  MoveL 5226 to (-61.59, 2.74, -134.54) mm, rotated rx -172.19 ry 6.28 rz 7.52 deg; joints [-5.137, -27.027, 87, 93.373, 104.768, 50.925, -36.259]
  MoveL 5227 to (-61.07, 2.44, -134.84) mm, rotated rx -172.19 ry 6.28 rz 7.52 deg; joints [-5.158, -27.049, 87.032, 93.353, 104.779, 50.915, -36.259]
  MoveL 5228 to (-60.98, 2.39, -135) mm, rotated rx -172.19 ry 6.28 rz 7.52 deg; joints [-5.162, -27.056, 87.036, 93.35, 104.781, 50.918, -36.259]
  MoveL 5229 to (-61.28, 2.57, -135.03) mm, rotated rx -172.19 ry 6.28 rz 7.52 deg; joints [-5.153, -27.051, 87.016, 93.362, 104.775, 50.934, -36.259]
  MoveL 5230 to (-61.68, 2.81, -135.05) mm, rotated rx -172.19 ry 6.28 rz 7.52 deg; joints [-5.14, -27.044, 86.989, 93.378, 104.768, 50.954, -36.259]
  MoveL 5231 to (-62.08, 3.07, -135.08) mm, rotated rx -172.19 ry 6.28 rz 7.52 deg; joints [-5.127, -27.036, 86.96, 93.395, 104.76, 50.975, -36.259]
  MoveL 5232 to (-62.45, 3.33, -135.14) mm, rotated rx -172.19 ry 6.28 rz 7.52 deg; joints [-5.115, -27.029, 86.931, 93.411, 104.753, 50.997, -36.259]
  MoveL 5233 to (-62.84, 3.58, -135.18) mm, rotated rx -172.19 ry 6.28 rz 7.52 deg; joints [-5.103, -27.021, 86.902, 93.427, 104.745, 51.019, -36.259]
  MoveL 5234 to (-63.26, 3.84, -135.2) mm, rotated rx -172.19 ry 6.28 rz 7.52 deg; joints [-5.089, -27.013, 86.874, 93.444, 104.737, 51.04, -36.259]
  MoveL 5235 to (-65.52, 5.16, -135.2) mm, rotated rx -172.19 ry 6.28 rz 7.52 deg; joints [-5.015, -26.97, 86.726, 93.535, 104.693, 51.145, -36.259]
  MoveL 5236 to (-65.91, 5.4, -135.22) mm, rotated rx -172.19 ry 6.28 rz 7.52 deg; joints [-5.002, -26.962, 86.699, 93.551, 104.686, 51.165, -36.259]
  MoveL 5237 to (-66.23, 5.62, -135.26) mm, rotated rx -172.19 ry 6.28 rz 7.52 deg; joints [-4.992, -26.956, 86.674, 93.565, 104.68, 51.183, -36.259]
  MoveL 5238 to (-66.62, 5.86, -135.28) mm, rotated rx -172.19 ry 6.28 rz 7.52 deg; joints [-4.979, -26.948, 86.646, 93.581, 104.672, 51.203, -36.259]
  MoveL 5239 to (-67.12, 6.18, -135.3) mm, rotated rx -172.19 ry 6.28 rz 7.52 deg; joints [-4.963, -26.938, 86.611, 93.601, 104.662, 51.229, -36.259]
  MoveL 5240 to (-67.73, 6.57, -135.35) mm, rotated rx -172.19 ry 6.28 rz 7.52 deg; joints [-4.944, -26.925, 86.566, 93.626, 104.65, 51.262, -36.259]
  MoveL 5241 to (-68.25, 6.9, -135.38) mm, rotated rx -172.19 ry 6.28 rz 7.52 deg; joints [-4.927, -26.915, 86.529, 93.648, 104.64, 51.289, -36.259]
  MoveL 5242 to (-68.71, 7.17, -135.38) mm, rotated rx -172.19 ry 6.28 rz 7.52 deg; joints [-4.912, -26.906, 86.498, 93.666, 104.631, 51.311, -36.259]
  MoveL 5243 to (-70.07, 7.96, -135.38) mm, rotated rx -172.19 ry 6.28 rz 7.52 deg; joints [-4.867, -26.879, 86.409, 93.721, 104.605, 51.374, -36.259]
  MoveL 5244 to (-72.42, 9.68, -135.73) mm, rotated rx -172.19 ry 6.28 rz 7.52 deg; joints [-4.794, -26.827, 86.213, 93.82, 104.558, 51.518, -36.259]
  MoveL 5245 to (-73.31, 10.62, -136.15) mm, rotated rx -172.19 ry 6.28 rz 7.52 deg; joints [-4.77, -26.801, 86.105, 93.862, 104.54, 51.603, -36.259]
  MoveL 5246 to (-74.01, 11.62, -136.75) mm, rotated rx -172.19 ry 6.28 rz 7.52 deg; joints [-4.754, -26.775, 85.989, 93.899, 104.526, 51.696, -36.259]
  MoveL 5247 to (-74.82, 13.8, -138.46) mm, rotated rx -172.19 ry 6.28 rz 7.52 deg; joints [-4.747, -26.726, 85.735, 93.958, 104.508, 51.906, -36.259]
  MoveL 5248 to (-74.85, 16.21, -140.86) mm, rotated rx -172.19 ry 6.28 rz 7.52 deg; joints [-4.773, -26.678, 85.452, 93.996, 104.506, 52.149, -36.259]
  MoveL 5249 to (-74.23, 18.17, -143.26) mm, rotated rx -172.19 ry 6.28 rz 7.52 deg; joints [-4.821, -26.645, 85.218, 94.008, 104.516, 52.358, -36.259]
  MoveL 5250 to (-73.72, 18.73, -144.2) mm, rotated rx -172.19 ry 6.28 rz 7.52 deg; joints [-4.848, -26.641, 85.15, 94.001, 104.526, 52.425, -36.259]
  MoveL 5251 to (-73.07, 19.02, -144.97) mm, rotated rx -172.19 ry 6.28 rz 7.52 deg; joints [-4.878, -26.644, 85.114, 93.986, 104.539, 52.467, -36.259]
  MoveL 5252 to (-72.69, 19.06, -145.29) mm, rotated rx -172.19 ry 6.28 rz 7.52 deg; joints [-4.894, -26.649, 85.108, 93.976, 104.547, 52.478, -36.259]
  MoveL 5253 to (-72.28, 19.03, -145.57) mm, rotated rx -172.19 ry 6.28 rz 7.52 deg; joints [-4.91, -26.656, 85.111, 93.963, 104.555, 52.483, -36.259]
  MoveL 5254 to (-71.36, 18.75, -145.99) mm, rotated rx -172.19 ry 6.28 rz 7.52 deg; joints [-4.945, -26.675, 85.14, 93.931, 104.574, 52.475, -36.259]
  MoveL 5255 to (-70.31, 18.2, -146.25) mm, rotated rx -172.19 ry 6.28 rz 7.52 deg; joints [-4.982, -26.702, 85.201, 93.891, 104.595, 52.441, -36.259]
  MoveL 5256 to (-69.12, 17.37, -146.34) mm, rotated rx -172.19 ry 6.28 rz 7.52 deg; joints [-5.022, -26.738, 85.295, 93.842, 104.62, 52.381, -36.259]
  MoveL 5257 to (-68.7, 17.06, -146.34) mm, rotated rx -172.19 ry 6.28 rz 7.52 deg; joints [-5.036, -26.75, 85.332, 93.824, 104.629, 52.358, -36.259]
  MoveL 5258 to (-68.38, 16.76, -146.28) mm, rotated rx -172.19 ry 6.28 rz 7.52 deg; joints [-5.046, -26.761, 85.366, 93.81, 104.636, 52.334, -36.259]
  MoveL 5259 to (-68.06, 16.46, -146.22) mm, rotated rx -172.19 ry 6.28 rz 7.52 deg; joints [-5.056, -26.772, 85.4, 93.795, 104.642, 52.31, -36.259]
  MoveL 5260 to (-67.7, 16.15, -146.18) mm, rotated rx -172.19 ry 6.28 rz 7.52 deg; joints [-5.067, -26.784, 85.435, 93.779, 104.65, 52.286, -36.259]
  MoveL 5261 to (-67.32, 15.84, -146.17) mm, rotated rx -172.19 ry 6.28 rz 7.52 deg; joints [-5.079, -26.796, 85.471, 93.763, 104.658, 52.263, -36.259]
  MoveL 5262 to (-66.9, 15.51, -146.16) mm, rotated rx -172.19 ry 6.28 rz 7.52 deg; joints [-5.093, -26.809, 85.508, 93.745, 104.666, 52.238, -36.259]
  MoveL 5263 to (-66.48, 15.19, -146.16) mm, rotated rx -172.19 ry 6.28 rz 7.52 deg; joints [-5.107, -26.822, 85.544, 93.727, 104.675, 52.215, -36.259]
  MoveL 5264 to (-66.07, 14.89, -146.18) mm, rotated rx -172.19 ry 6.28 rz 7.52 deg; joints [-5.12, -26.834, 85.578, 93.71, 104.683, 52.193, -36.259]
  MoveL 5265 to (-65.67, 14.6, -146.19) mm, rotated rx -172.19 ry 6.28 rz 7.52 deg; joints [-5.134, -26.846, 85.611, 93.693, 104.692, 52.171, -36.259]
  MoveL 5266 to (-65.31, 14.31, -146.17) mm, rotated rx -172.19 ry 6.28 rz 7.52 deg; joints [-5.145, -26.857, 85.644, 93.678, 104.699, 52.149, -36.259]
  MoveL 5267 to (-64.96, 14, -146.13) mm, rotated rx -172.19 ry 6.28 rz 7.52 deg; joints [-5.156, -26.868, 85.678, 93.662, 104.706, 52.126, -36.259]
  MoveL 5268 to (-64.55, 13.65, -146.08) mm, rotated rx -172.19 ry 6.28 rz 7.52 deg; joints [-5.169, -26.881, 85.719, 93.644, 104.715, 52.098, -36.259]
  MoveL 5269 to (-64.02, 13.18, -146.02) mm, rotated rx -172.19 ry 6.28 rz 7.52 deg; joints [-5.186, -26.899, 85.772, 93.621, 104.726, 52.062, -36.259]
  MoveL 5270 to (-63.52, 12.77, -146) mm, rotated rx -172.19 ry 6.28 rz 7.52 deg; joints [-5.202, -26.915, 85.818, 93.599, 104.736, 52.031, -36.259]
  MoveL 5271 to (-61.45, 11.18, -146) mm, rotated rx -172.19 ry 6.28 rz 7.52 deg; joints [-5.27, -26.978, 85.997, 93.511, 104.778, 51.913, -36.259]
  MoveL 5272 to (-60.96, 10.78, -145.96) mm, rotated rx -172.19 ry 6.28 rz 7.52 deg; joints [-5.286, -26.992, 86.042, 93.49, 104.788, 51.883, -36.259]
  MoveL 5273 to (-60.54, 10.42, -145.9) mm, rotated rx -172.19 ry 6.28 rz 7.52 deg; joints [-5.299, -27.005, 86.083, 93.471, 104.797, 51.854, -36.259]
  MoveL 5274 to (-60.38, 10.28, -145.76) mm, rotated rx -172.19 ry 6.28 rz 7.52 deg; joints [-5.303, -27.005, 86.099, 93.464, 104.799, 51.838, -36.259]
  MoveL 5275 to (-60.48, 10.36, -145.49) mm, rotated rx -172.19 ry 6.28 rz 7.52 deg; joints [-5.297, -26.992, 86.092, 93.467, 104.797, 51.831, -36.259]
  MoveL 5276 to (-60.82, 10.66, -145.09) mm, rotated rx -172.19 ry 6.28 rz 7.52 deg; joints [-5.281, -26.964, 86.061, 93.481, 104.788, 51.834, -36.259]
  MoveL 5277 to (-61.16, 9.69, -144.28) mm, rotated rx -172.19 ry 6.28 rz 7.52 deg; joints [-5.261, -26.994, 86.173, 93.477, 104.783, 51.749, -36.259]
  MoveL 5278 to (-60.58, 7.8, -144.07) mm, rotated rx -172.19 ry 6.28 rz 7.52 deg; joints [-5.278, -27.086, 86.384, 93.431, 104.799, 51.626, -36.259]
  MoveL 5279 to (-59.97, 5.89, -143.91) mm, rotated rx -172.19 ry 6.28 rz 7.52 deg; joints [-5.297, -27.181, 86.596, 93.384, 104.815, 51.506, -36.259]
  MoveL 5280 to (-59.34, 3.93, -143.75) mm, rotated rx -172.19 ry 6.28 rz 7.52 deg; joints [-5.316, -27.277, 86.813, 93.335, 104.832, 51.382, -36.259]
  MoveL 5281 to (-58.78, 2.14, -143.46) mm, rotated rx -172.19 ry 6.28 rz 7.52 deg; joints [-5.332, -27.359, 87.011, 93.291, 104.847, 51.263, -36.259]
  MoveL 5282 to (-58.13, 0.13, -143.27) mm, rotated rx -172.19 ry 6.28 rz 7.52 deg; joints [-5.352, -27.457, 87.232, 93.241, 104.864, 51.136, -36.259]
  MoveL 5283 to (-57.45, -1.98, -143.09) mm, rotated rx -172.19 ry 6.28 rz 7.52 deg; joints [-5.373, -27.559, 87.463, 93.189, 104.882, 51.003, -36.259]
  MoveL 5284 to (-56.75, -4.11, -143) mm, rotated rx -172.19 ry 6.28 rz 7.52 deg; joints [-5.396, -27.665, 87.696, 93.136, 104.9, 50.873, -36.259]
  MoveL 5285 to (-55.89, -6.7, -142.91) mm, rotated rx -172.19 ry 6.28 rz 7.52 deg; joints [-5.425, -27.795, 87.978, 93.071, 104.923, 50.717, -36.259]
  MoveL 5286 to (-55.27, -8.56, -142.81) mm, rotated rx -172.19 ry 6.28 rz 7.52 deg; joints [-5.445, -27.886, 88.18, 93.024, 104.939, 50.603, -36.259]
  MoveL 5287 to (-54.69, -10.29, -142.59) mm, rotated rx -172.19 ry 6.28 rz 7.52 deg; joints [-5.462, -27.966, 88.368, 92.98, 104.953, 50.491, -36.259]
  MoveL 5288 to (-54.05, -12.2, -142.4) mm, rotated rx -172.19 ry 6.28 rz 7.52 deg; joints [-5.482, -28.056, 88.576, 92.931, 104.969, 50.37, -36.259]
  MoveL 5289 to (-53.36, -14.22, -142.28) mm, rotated rx -172.19 ry 6.28 rz 7.52 deg; joints [-5.505, -28.154, 88.794, 92.88, 104.986, 50.246, -36.259]
  MoveL 5290 to (-52.68, -16.22, -142.1) mm, rotated rx -172.19 ry 6.28 rz 7.52 deg; joints [-5.526, -28.248, 89.01, 92.829, 105.003, 50.121, -36.259]
  MoveL 5291 to (-52, -18.22, -141.98) mm, rotated rx -172.19 ry 6.28 rz 7.52 deg; joints [-5.549, -28.344, 89.224, 92.777, 105.019, 49.999, -36.259]
  MoveL 5292 to (-51.29, -20.28, -141.8) mm, rotated rx -172.19 ry 6.28 rz 7.52 deg; joints [-5.571, -28.44, 89.445, 92.724, 105.036, 49.87, -36.259]
  MoveL 5293 to (-50.59, -22.3, -141.68) mm, rotated rx -172.19 ry 6.28 rz 7.52 deg; joints [-5.594, -28.537, 89.661, 92.672, 105.053, 49.748, -36.259]
  MoveL 5294 to (-49.88, -24.31, -141.45) mm, rotated rx -172.19 ry 6.28 rz 7.52 deg; joints [-5.617, -28.628, 89.876, 92.62, 105.069, 49.619, -36.259]
  MoveL 5295 to (-49.18, -26.33, -141.34) mm, rotated rx -172.19 ry 6.28 rz 7.52 deg; joints [-5.64, -28.724, 90.091, 92.567, 105.086, 49.497, -36.259]
  MoveL 5296 to (-48.48, -28.35, -141.22) mm, rotated rx -172.19 ry 6.28 rz 7.52 deg; joints [-5.663, -28.819, 90.305, 92.515, 105.102, 49.375, -36.259]
  MoveL 5297 to (-47.75, -30.36, -141) mm, rotated rx -172.19 ry 6.28 rz 7.52 deg; joints [-5.686, -28.909, 90.518, 92.462, 105.119, 49.248, -36.259]
  MoveL 5298 to (-47.05, -32.16, -140.8) mm, rotated rx -172.19 ry 6.28 rz 7.52 deg; joints [-5.709, -28.989, 90.71, 92.412, 105.134, 49.133, -36.259]
  MoveL 5299 to (-46.35, -33.78, -140.51) mm, rotated rx -172.19 ry 6.28 rz 7.52 deg; joints [-5.73, -29.055, 90.882, 92.365, 105.148, 49.024, -36.259]
  MoveL 5300 to (-45.62, -35.24, -140.1) mm, rotated rx -172.19 ry 6.28 rz 7.52 deg; joints [-5.75, -29.108, 91.038, 92.319, 105.162, 48.918, -36.259]
  MoveL 5301 to (-45.58, -33.75, -139.17) mm, rotated rx -172.19 ry 6.28 rz 7.52 deg; joints [-5.74, -28.991, 90.888, 92.337, 105.156, 48.951, -36.259]
  MoveL 5302 to (-45.51, -34.33, -139.16) mm, rotated rx -172.19 ry 6.28 rz 7.52 deg; joints [-5.743, -29.021, 90.948, 92.326, 105.159, 48.92, -36.259]
  MoveL 5303 to (-45.48, -34.86, -139.14) mm, rotated rx -172.19 ry 6.28 rz 7.52 deg; joints [-5.744, -29.048, 91.004, 92.318, 105.16, 48.89, -36.259]
  MoveL 5304 to (-45.5, -35.33, -139.08) mm, rotated rx -172.19 ry 6.28 rz 7.52 deg; joints [-5.743, -29.071, 91.053, 92.311, 105.161, 48.863, -36.259]
  MoveL 5305 to (-45.54, -35.78, -139.01) mm, rotated rx -172.19 ry 6.28 rz 7.52 deg; joints [-5.741, -29.093, 91.1, 92.306, 105.161, 48.837, -36.259]
  MoveL 5306 to (-45.62, -36.23, -138.96) mm, rotated rx -172.19 ry 6.28 rz 7.52 deg; joints [-5.738, -29.117, 91.149, 92.302, 105.161, 48.812, -36.259]
  MoveL 5307 to (-45.72, -36.71, -138.93) mm, rotated rx -172.19 ry 6.28 rz 7.52 deg; joints [-5.734, -29.143, 91.198, 92.299, 105.16, 48.787, -36.259]
  MoveL 5308 to (-45.85, -37.22, -138.91) mm, rotated rx -172.19 ry 6.28 rz 7.52 deg; joints [-5.73, -29.172, 91.252, 92.296, 105.159, 48.761, -36.259]
  MoveL 5309 to (-45.98, -37.73, -138.91) mm, rotated rx -172.19 ry 6.28 rz 7.52 deg; joints [-5.726, -29.201, 91.305, 92.293, 105.158, 48.737, -36.259]
  MoveL 5310 to (-46.1, -38.18, -138.9) mm, rotated rx -172.19 ry 6.28 rz 7.52 deg; joints [-5.722, -29.227, 91.352, 92.291, 105.157, 48.714, -36.259]
  MoveL 5311 to (-46.19, -38.6, -138.88) mm, rotated rx -172.19 ry 6.28 rz 7.52 deg; joints [-5.719, -29.249, 91.396, 92.288, 105.156, 48.693, -36.259]
  MoveL 5312 to (-46.3, -39.06, -138.86) mm, rotated rx -172.19 ry 6.28 rz 7.52 deg; joints [-5.715, -29.276, 91.444, 92.285, 105.156, 48.669, -36.259]
  MoveL 5313 to (-46.44, -39.57, -138.86) mm, rotated rx -172.19 ry 6.28 rz 7.52 deg; joints [-5.711, -29.305, 91.497, 92.282, 105.155, 48.645, -36.259]
  MoveL 5314 to (-46.59, -40.16, -138.84) mm, rotated rx -172.19 ry 6.28 rz 7.52 deg; joints [-5.706, -29.338, 91.559, 92.279, 105.153, 48.615, -36.259]
  MoveL 5315 to (-46.75, -40.84, -138.8) mm, rotated rx -172.19 ry 6.28 rz 7.52 deg; joints [-5.7, -29.375, 91.63, 92.275, 105.152, 48.58, -36.259]
  MoveL 5316 to (-46.9, -41.43, -138.78) mm, rotated rx -172.19 ry 6.28 rz 7.52 deg; joints [-5.696, -29.408, 91.691, 92.271, 105.151, 48.551, -36.259]
  MoveL 5317 to (-47.05, -42.05, -138.76) mm, rotated rx -172.19 ry 6.28 rz 7.52 deg; joints [-5.691, -29.443, 91.756, 92.268, 105.15, 48.52, -36.259]
  MoveL 5318 to (-47.2, -42.75, -138.72) mm, rotated rx -172.19 ry 6.28 rz 7.52 deg; joints [-5.685, -29.481, 91.828, 92.263, 105.149, 48.484, -36.259]
  MoveL 5319 to (-47.35, -43.32, -138.7) mm, rotated rx -172.19 ry 6.28 rz 7.52 deg; joints [-5.681, -29.513, 91.888, 92.26, 105.148, 48.456, -36.259]
  MoveL 5320 to (-47.49, -43.84, -138.7) mm, rotated rx -172.19 ry 6.28 rz 7.52 deg; joints [-5.676, -29.543, 91.942, 92.257, 105.147, 48.43, -36.259]
  MoveL 5321 to (-47.9, -45.36, -138.7) mm, rotated rx -172.19 ry 6.28 rz 7.52 deg; joints [-5.663, -29.631, 92.099, 92.25, 105.143, 48.358, -36.259]
  MoveL 5322 to (-48.35, -46.74, -138.79) mm, rotated rx -172.19 ry 6.28 rz 7.52 deg; joints [-5.65, -29.714, 92.241, 92.246, 105.139, 48.297, -36.259]
  MoveL 5323 to (-48.86, -47.82, -139.04) mm, rotated rx -172.19 ry 6.28 rz 7.52 deg; joints [-5.636, -29.789, 92.351, 92.249, 105.134, 48.261, -36.259]
  MoveL 5324 to (-49.43, -48.59, -139.46) mm, rotated rx -172.19 ry 6.28 rz 7.52 deg; joints [-5.622, -29.855, 92.427, 92.258, 105.128, 48.25, -36.259]
  MoveL 5325 to (-49.73, -48.86, -139.73) mm, rotated rx -172.19 ry 6.28 rz 7.52 deg; joints [-5.615, -29.885, 92.453, 92.265, 105.125, 48.254, -36.259]
  MoveL 5326 to (-50.05, -49.05, -140.05) mm, rotated rx -172.19 ry 6.28 rz 7.52 deg; joints [-5.608, -29.913, 92.471, 92.274, 105.121, 48.264, -36.259]
  MoveL 5327 to (-50.74, -49.22, -140.81) mm, rotated rx -172.19 ry 6.28 rz 7.52 deg; joints [-5.594, -29.961, 92.483, 92.297, 105.113, 48.302, -36.259]
  MoveL 5328 to (-51.49, -49.08, -141.74) mm, rotated rx -172.19 ry 6.28 rz 7.52 deg; joints [-5.579, -30.001, 92.462, 92.326, 105.104, 48.365, -36.259]
  MoveL 5329 to (-53.16, -47.88, -144.1) mm, rotated rx -172.19 ry 6.28 rz 7.52 deg; joints [-5.55, -30.055, 92.321, 92.404, 105.083, 48.565, -36.259]
  MoveL 5330 to (-54.58, -45.94, -146.46) mm, rotated rx -172.19 ry 6.28 rz 7.52 deg; joints [-5.529, -30.063, 92.103, 92.484, 105.063, 48.799, -36.259]
  MoveL 5331 to (-55.24, -43.71, -148.15) mm, rotated rx -172.19 ry 6.28 rz 7.52 deg; joints [-5.525, -30.018, 91.86, 92.54, 105.053, 49.005, -36.259]
  MoveL 5332 to (-55.29, -42.49, -148.74) mm, rotated rx -172.19 ry 6.28 rz 7.52 deg; joints [-5.53, -29.976, 91.729, 92.56, 105.051, 49.096, -36.259]
  MoveL 5333 to (-55.15, -41.2, -149.16) mm, rotated rx -172.19 ry 6.28 rz 7.52 deg; joints [-5.539, -29.921, 91.592, 92.574, 105.051, 49.181, -36.259]
  MoveL 5334 to (-54.3, -38.41, -149.5) mm, rotated rx -172.19 ry 6.28 rz 7.52 deg; joints [-5.57, -29.771, 91.3, 92.585, 105.06, 49.329, -36.259]
  MoveL 5335 to (-52.69, -34.55, -149.5) mm, rotated rx -172.19 ry 6.28 rz 7.52 deg; joints [-5.622, -29.537, 90.897, 92.585, 105.077, 49.505, -36.259]
  MoveL 5336 to (-52.49, -34.03, -149.52) mm, rotated rx -172.19 ry 6.28 rz 7.52 deg; joints [-5.628, -29.507, 90.843, 92.586, 105.079, 49.53, -36.259]
  MoveL 5337 to (-52.32, -33.54, -149.56) mm, rotated rx -172.19 ry 6.28 rz 7.52 deg; joints [-5.634, -29.479, 90.791, 92.587, 105.081, 49.555, -36.259]
  MoveL 5338 to (-52.15, -33.03, -149.62) mm, rotated rx -172.19 ry 6.28 rz 7.52 deg; joints [-5.64, -29.452, 90.737, 92.589, 105.083, 49.582, -36.259]
  MoveL 5339 to (-52.01, -32.53, -149.7) mm, rotated rx -172.19 ry 6.28 rz 7.52 deg; joints [-5.646, -29.426, 90.685, 92.591, 105.084, 49.61, -36.259]
  MoveL 5340 to (-51.87, -32.05, -149.78) mm, rotated rx -172.19 ry 6.28 rz 7.52 deg; joints [-5.651, -29.4, 90.633, 92.594, 105.085, 49.637, -36.259]
  MoveL 5341 to (-51.71, -31.59, -149.82) mm, rotated rx -172.19 ry 6.28 rz 7.52 deg; joints [-5.657, -29.374, 90.585, 92.595, 105.087, 49.66, -36.259]
  MoveL 5342 to (-51.53, -31.14, -149.84) mm, rotated rx -172.19 ry 6.28 rz 7.52 deg; joints [-5.663, -29.348, 90.538, 92.595, 105.089, 49.681, -36.259]
  MoveL 5343 to (-51.33, -30.66, -149.84) mm, rotated rx -172.19 ry 6.28 rz 7.52 deg; joints [-5.669, -29.318, 90.487, 92.595, 105.091, 49.704, -36.259]
  MoveL 5344 to (-51.11, -30.07, -149.87) mm, rotated rx -172.19 ry 6.28 rz 7.52 deg; joints [-5.677, -29.285, 90.425, 92.596, 105.093, 49.733, -36.259]
  MoveL 5345 to (-50.88, -29.43, -149.93) mm, rotated rx -172.19 ry 6.28 rz 7.52 deg; joints [-5.685, -29.248, 90.357, 92.598, 105.096, 49.766, -36.259]
  MoveL 5346 to (-50.69, -28.86, -149.95) mm, rotated rx -172.19 ry 6.28 rz 7.52 deg; joints [-5.691, -29.216, 90.298, 92.6, 105.098, 49.793, -36.259]
  MoveL 5347 to (-50.55, -28.33, -149.96) mm, rotated rx -172.19 ry 6.28 rz 7.52 deg; joints [-5.695, -29.184, 90.241, 92.603, 105.099, 49.82, -36.259]
  MoveL 5348 to (-50.45, -27.78, -149.96) mm, rotated rx -172.19 ry 6.28 rz 7.52 deg; joints [-5.698, -29.153, 90.184, 92.607, 105.099, 49.847, -36.259]
  MoveL 5349 to (-50.48, -27.21, -149.96) mm, rotated rx -172.19 ry 6.28 rz 7.52 deg; joints [-5.697, -29.122, 90.123, 92.616, 105.097, 49.878, -36.259]
  MoveL 5350 to (-50.57, -26.6, -149.96) mm, rotated rx -172.19 ry 6.28 rz 7.52 deg; joints [-5.694, -29.09, 90.059, 92.628, 105.094, 49.911, -36.259]
  MoveL 5351 to (-50.69, -28.17, -150.92) mm, rotated rx -172.19 ry 6.28 rz 7.52 deg; joints [-5.702, -29.215, 90.218, 92.612, 105.099, 49.876, -36.259]
  MoveL 5352 to (-51.15, -27.02, -151.34) mm, rotated rx -172.19 ry 6.28 rz 7.52 deg; joints [-5.69, -29.174, 90.092, 92.644, 105.09, 49.963, -36.259]
  MoveL 5353 to (-51.58, -25.67, -151.67) mm, rotated rx -172.19 ry 6.28 rz 7.52 deg; joints [-5.679, -29.119, 89.947, 92.678, 105.08, 50.056, -36.259]
  MoveL 5354 to (-51.99, -24.11, -151.92) mm, rotated rx -172.19 ry 6.28 rz 7.52 deg; joints [-5.667, -29.048, 89.78, 92.715, 105.07, 50.156, -36.259]
  MoveL 5355 to (-52.43, -22.02, -152.03) mm, rotated rx -172.19 ry 6.28 rz 7.52 deg; joints [-5.653, -28.944, 89.557, 92.759, 105.057, 50.277, -36.259]
  MoveL 5356 to (-52.89, -19.94, -152.26) mm, rotated rx -172.19 ry 6.28 rz 7.52 deg; joints [-5.639, -28.844, 89.334, 92.804, 105.045, 50.405, -36.259]
  MoveL 5357 to (-53.32, -17.86, -152.38) mm, rotated rx -172.19 ry 6.28 rz 7.52 deg; joints [-5.625, -28.739, 89.11, 92.848, 105.032, 50.527, -36.259]
  MoveL 5358 to (-53.75, -15.77, -152.49) mm, rotated rx -172.19 ry 6.28 rz 7.52 deg; joints [-5.611, -28.633, 88.886, 92.892, 105.019, 50.649, -36.259]
  MoveL 5359 to (-54.19, -13.68, -152.73) mm, rotated rx -172.19 ry 6.28 rz 7.52 deg; joints [-5.598, -28.532, 88.66, 92.937, 105.006, 50.778, -36.259]
  MoveL 5360 to (-54.62, -11.59, -152.85) mm, rotated rx -172.19 ry 6.28 rz 7.52 deg; joints [-5.584, -28.426, 88.434, 92.981, 104.993, 50.901, -36.259]
  MoveL 5361 to (-55.04, -9.5, -152.97) mm, rotated rx -172.19 ry 6.28 rz 7.52 deg; joints [-5.57, -28.319, 88.208, 93.024, 104.98, 51.024, -36.259]
  MoveL 5362 to (-55.53, -7.09, -153.13) mm, rotated rx -172.19 ry 6.28 rz 7.52 deg; joints [-5.554, -28.197, 87.946, 93.075, 104.964, 51.168, -36.259]
  MoveL 5363 to (-55.94, -5.03, -153.32) mm, rotated rx -172.19 ry 6.28 rz 7.52 deg; joints [-5.542, -28.094, 87.722, 93.118, 104.952, 51.294, -36.259]
  MoveL 5364 to (-56.39, -2.76, -153.52) mm, rotated rx -172.19 ry 6.28 rz 7.52 deg; joints [-5.528, -27.98, 87.474, 93.165, 104.937, 51.431, -36.259]
  MoveL 5365 to (-56.82, -0.54, -153.77) mm, rotated rx -172.19 ry 6.28 rz 7.52 deg; joints [-5.516, -27.87, 87.23, 93.212, 104.924, 51.569, -36.259]
  MoveL 5366 to (-57.23, 1.55, -153.89) mm, rotated rx -172.19 ry 6.28 rz 7.52 deg; joints [-5.503, -27.761, 87.001, 93.255, 104.91, 51.694, -36.259]
  MoveL 5367 to (-57.65, 3.64, -153.89) mm, rotated rx -172.19 ry 6.28 rz 7.52 deg; joints [-5.488, -27.648, 86.771, 93.298, 104.896, 51.814, -36.259]
  MoveL 5368 to (-58.05, 5.71, -153.97) mm, rotated rx -172.19 ry 6.28 rz 7.52 deg; joints [-5.475, -27.539, 86.544, 93.341, 104.882, 51.935, -36.259]
  MoveL 5369 to (-58.42, 7.73, -154.18) mm, rotated rx -172.19 ry 6.28 rz 7.52 deg; joints [-5.464, -27.436, 86.319, 93.382, 104.87, 52.061, -36.259]
  MoveL 5370 to (-58.81, 10, -154.54) mm, rotated rx -172.19 ry 6.28 rz 7.52 deg; joints [-5.454, -27.325, 86.066, 93.428, 104.856, 52.207, -36.259]
  MoveL 5371 to (-59.12, 11.78, -154.75) mm, rotated rx -172.19 ry 6.28 rz 7.52 deg; joints [-5.446, -27.235, 85.868, 93.464, 104.845, 52.319, -36.259]
  MoveL 5372 to (-59.52, 14.2, -155.04) mm, rotated rx -172.19 ry 6.28 rz 7.52 deg; joints [-5.435, -27.112, 85.597, 93.512, 104.831, 52.471, -36.259]
  MoveL 5373 to (-59.92, 16.38, -155.15) mm, rotated rx -172.19 ry 6.28 rz 7.52 deg; joints [-5.422, -26.996, 85.354, 93.557, 104.816, 52.601, -36.259]
  MoveL 5374 to (-60.33, 18.46, -155.16) mm, rotated rx -172.19 ry 6.28 rz 7.52 deg; joints [-5.408, -26.881, 85.121, 93.6, 104.801, 52.723, -36.259]
  MoveL 5375 to (-59.99, 19.29, -155.95) mm, rotated rx -172.19 ry 6.28 rz 7.52 deg; joints [-5.428, -26.858, 85.024, 93.602, 104.807, 52.8, -36.259]
  MoveL 5376 to (-59.74, 18.92, -156.34) mm, rotated rx -172.19 ry 6.28 rz 7.52 deg; joints [-5.441, -26.89, 85.061, 93.59, 104.814, 52.795, -36.259]
  MoveL 5377 to (-59.67, 18.8, -156.59) mm, rotated rx -172.19 ry 6.28 rz 7.52 deg; joints [-5.446, -26.905, 85.073, 93.587, 104.817, 52.798, -36.259]
  MoveL 5378 to (-59.77, 18.91, -156.71) mm, rotated rx -172.19 ry 6.28 rz 7.52 deg; joints [-5.444, -26.905, 85.06, 93.592, 104.815, 52.811, -36.259]
  MoveL 5379 to (-60.03, 19.19, -156.73) mm, rotated rx -172.19 ry 6.28 rz 7.52 deg; joints [-5.435, -26.892, 85.028, 93.604, 104.809, 52.832, -36.259]
  MoveL 5380 to (-60.36, 19.53, -156.74) mm, rotated rx -172.19 ry 6.28 rz 7.52 deg; joints [-5.425, -26.877, 84.989, 93.619, 104.802, 52.856, -36.259]
  MoveL 5381 to (-61.47, 20.64, -156.74) mm, rotated rx -172.19 ry 6.28 rz 7.52 deg; joints [-5.388, -26.828, 84.864, 93.67, 104.778, 52.933, -36.259]
  MoveL 5382 to (-61.85, 21.04, -156.76) mm, rotated rx -172.19 ry 6.28 rz 7.52 deg; joints [-5.376, -26.811, 84.818, 93.688, 104.77, 52.961, -36.259]
  MoveL 5383 to (-62.22, 21.45, -156.81) mm, rotated rx -172.19 ry 6.28 rz 7.52 deg; joints [-5.364, -26.793, 84.772, 93.705, 104.762, 52.992, -36.259]
  MoveL 5384 to (-62.59, 21.9, -156.89) mm, rotated rx -172.19 ry 6.28 rz 7.52 deg; joints [-5.353, -26.775, 84.721, 93.723, 104.754, 53.025, -36.259]
  MoveL 5385 to (-62.95, 22.31, -156.95) mm, rotated rx -172.19 ry 6.28 rz 7.52 deg; joints [-5.342, -26.758, 84.673, 93.741, 104.746, 53.056, -36.259]
  MoveL 5386 to (-63.31, 22.7, -156.97) mm, rotated rx -172.19 ry 6.28 rz 7.52 deg; joints [-5.33, -26.741, 84.629, 93.758, 104.738, 53.084, -36.259]
  MoveL 5387 to (-63.65, 23.06, -156.99) mm, rotated rx -172.19 ry 6.28 rz 7.52 deg; joints [-5.319, -26.726, 84.588, 93.774, 104.73, 53.11, -36.259]
  MoveL 5388 to (-63.95, 23.41, -157.04) mm, rotated rx -172.19 ry 6.28 rz 7.52 deg; joints [-5.31, -26.711, 84.548, 93.788, 104.724, 53.135, -36.259]
  MoveL 5389 to (-64.25, 23.74, -157.08) mm, rotated rx -172.19 ry 6.28 rz 7.52 deg; joints [-5.301, -26.697, 84.51, 93.802, 104.717, 53.16, -36.259]
  MoveL 5390 to (-64.59, 24.1, -157.09) mm, rotated rx -172.19 ry 6.28 rz 7.52 deg; joints [-5.29, -26.681, 84.469, 93.818, 104.71, 53.185, -36.259]
  MoveL 5391 to (-64.99, 24.52, -157.11) mm, rotated rx -172.19 ry 6.28 rz 7.52 deg; joints [-5.277, -26.662, 84.421, 93.837, 104.701, 53.215, -36.259]
  MoveL 5392 to (-65.46, 25.05, -157.16) mm, rotated rx -172.19 ry 6.28 rz 7.52 deg; joints [-5.262, -26.64, 84.36, 93.859, 104.69, 53.254, -36.259]
  MoveL 5393 to (-65.87, 25.49, -157.19) mm, rotated rx -172.19 ry 6.28 rz 7.52 deg; joints [-5.249, -26.62, 84.31, 93.878, 104.681, 53.286, -36.259]
  MoveL 5394 to (-67.36, 26.98, -157.2) mm, rotated rx -172.19 ry 6.28 rz 7.52 deg; joints [-5.2, -26.553, 84.14, 93.945, 104.648, 53.39, -36.259]
  MoveL 5395 to (-69.21, 29.23, -157.53) mm, rotated rx -172.19 ry 6.28 rz 7.52 deg; joints [-5.144, -26.457, 83.879, 94.035, 104.606, 53.557, -36.259]
  MoveL 5396 to (-69.83, 30.36, -157.94) mm, rotated rx -172.19 ry 6.28 rz 7.52 deg; joints [-5.128, -26.413, 83.746, 94.072, 104.592, 53.648, -36.259]
  MoveL 5397 to (-70.25, 31.5, -158.51) mm, rotated rx -172.19 ry 6.28 rz 7.52 deg; joints [-5.121, -26.373, 83.611, 94.102, 104.581, 53.745, -36.259]
  MoveL 5398 to (-70.5, 33.79, -160.16) mm, rotated rx -172.19 ry 6.28 rz 7.52 deg; joints [-5.131, -26.299, 83.337, 94.146, 104.572, 53.953, -36.259]
  MoveL 5399 to (-69.95, 36.11, -162.47) mm, rotated rx -172.19 ry 6.28 rz 7.52 deg; joints [-5.174, -26.237, 83.055, 94.167, 104.579, 54.182, -36.259]
  MoveL 5400 to (-68.87, 37.82, -164.78) mm, rotated rx -172.19 ry 6.28 rz 7.52 deg; joints [-5.234, -26.203, 82.84, 94.165, 104.599, 54.37, -36.259]
  MoveL 5401 to (-68.24, 38.23, -165.68) mm, rotated rx -172.19 ry 6.28 rz 7.52 deg; joints [-5.264, -26.203, 82.787, 94.154, 104.612, 54.425, -36.259]
  MoveL 5402 to (-67.55, 38.33, -166.42) mm, rotated rx -172.19 ry 6.28 rz 7.52 deg; joints [-5.294, -26.214, 82.77, 94.136, 104.627, 54.456, -36.259]
  MoveL 5403 to (-67.18, 38.27, -166.73) mm, rotated rx -172.19 ry 6.28 rz 7.52 deg; joints [-5.31, -26.224, 82.775, 94.124, 104.635, 54.461, -36.259]
  MoveL 5404 to (-66.8, 38.13, -167) mm, rotated rx -172.19 ry 6.28 rz 7.52 deg; joints [-5.325, -26.236, 82.789, 94.111, 104.643, 54.461, -36.259]
  MoveL 5405 to (-65.98, 37.63, -167.41) mm, rotated rx -172.19 ry 6.28 rz 7.52 deg; joints [-5.356, -26.27, 82.844, 94.08, 104.662, 54.44, -36.259]
  MoveL 5406 to (-65.1, 36.83, -167.66) mm, rotated rx -172.19 ry 6.28 rz 7.52 deg; joints [-5.387, -26.316, 82.935, 94.042, 104.682, 54.394, -36.259]
  MoveL 5407 to (-64.17, 35.72, -167.74) mm, rotated rx -172.19 ry 6.28 rz 7.52 deg; joints [-5.419, -26.372, 83.062, 93.998, 104.704, 54.322, -36.259]
  MoveL 5408 to (-61.93, 32.82, -167.74) mm, rotated rx -172.19 ry 6.28 rz 7.52 deg; joints [-5.492, -26.515, 83.396, 93.887, 104.758, 54.128, -36.259]
  MoveL 5409 to (-61.65, 32.45, -167.73) mm, rotated rx -172.19 ry 6.28 rz 7.52 deg; joints [-5.501, -26.533, 83.439, 93.873, 104.764, 54.103, -36.259]
  MoveL 5410 to (-61.42, 32.11, -167.7) mm, rotated rx -172.19 ry 6.28 rz 7.52 deg; joints [-5.508, -26.549, 83.478, 93.861, 104.77, 54.079, -36.259]
  MoveL 5411 to (-61.13, 31.73, -167.68) mm, rotated rx -172.19 ry 6.28 rz 7.52 deg; joints [-5.518, -26.567, 83.522, 93.847, 104.776, 54.053, -36.259]
  MoveL 5412 to (-58.89, 28.83, -167.68) mm, rotated rx -172.19 ry 6.28 rz 7.52 deg; joints [-5.591, -26.709, 83.854, 93.736, 104.829, 53.86, -36.259]
  MoveL 5413 to (-58.58, 28.39, -167.66) mm, rotated rx -172.19 ry 6.28 rz 7.52 deg; joints [-5.601, -26.73, 83.904, 93.719, 104.836, 53.83, -36.259]
  MoveL 5414 to (-58.29, 27.93, -167.63) mm, rotated rx -172.19 ry 6.28 rz 7.52 deg; joints [-5.61, -26.752, 83.957, 93.704, 104.843, 53.798, -36.259]
  MoveL 5415 to (-58.07, 27.49, -167.58) mm, rotated rx -172.19 ry 6.28 rz 7.52 deg; joints [-5.617, -26.773, 84.007, 93.69, 104.849, 53.769, -36.259]
  MoveL 5416 to (-57.94, 27.13, -167.52) mm, rotated rx -172.19 ry 6.28 rz 7.52 deg; joints [-5.621, -26.79, 84.048, 93.681, 104.853, 53.744, -36.259]
  MoveL 5417 to (-57.9, 26.94, -167.35) mm, rotated rx -172.19 ry 6.28 rz 7.52 deg; joints [-5.621, -26.794, 84.071, 93.677, 104.853, 53.725, -36.259]
  MoveL 5418 to (-57.93, 26.91, -167.02) mm, rotated rx -172.19 ry 6.28 rz 7.52 deg; joints [-5.616, -26.785, 84.077, 93.676, 104.852, 53.709, -36.259]
  MoveL 5419 to (-58.01, 27.05, -166.51) mm, rotated rx -172.19 ry 6.28 rz 7.52 deg; joints [-5.608, -26.76, 84.066, 93.679, 104.848, 53.694, -36.259]
  MoveL 5420 to (-58.52, 26.4, -165.05) mm, rotated rx -172.19 ry 6.28 rz 7.52 deg; joints [-5.575, -26.753, 84.152, 93.682, 104.837, 53.597, -36.259]
  MoveL 5421 to (-58.24, 22.14, -165.05) mm, rotated rx -172.19 ry 6.28 rz 7.52 deg; joints [-5.586, -26.998, 84.631, 93.611, 104.858, 53.356, -36.259]
  MoveL 5422 to (-58.11, 20.1, -165.01) mm, rotated rx -172.19 ry 6.28 rz 7.52 deg; joints [-5.591, -27.113, 84.859, 93.577, 104.867, 53.24, -36.259]
  MoveL 5423 to (-57.98, 18.13, -164.92) mm, rotated rx -172.19 ry 6.28 rz 7.52 deg; joints [-5.595, -27.223, 85.08, 93.544, 104.876, 53.125, -36.259]
  MoveL 5424 to (-57.86, 16.12, -164.83) mm, rotated rx -172.19 ry 6.28 rz 7.52 deg; joints [-5.6, -27.336, 85.305, 93.51, 104.885, 53.009, -36.259]
  MoveL 5425 to (-57.73, 14.15, -164.73) mm, rotated rx -172.19 ry 6.28 rz 7.52 deg; joints [-5.604, -27.444, 85.524, 93.478, 104.894, 52.894, -36.259]
  MoveL 5426 to (-57.62, 12.06, -164.69) mm, rotated rx -172.19 ry 6.28 rz 7.52 deg; joints [-5.608, -27.562, 85.756, 93.444, 104.904, 52.777, -36.259]
  MoveL 5427 to (-57.58, 9.86, -164.66) mm, rotated rx -172.19 ry 6.28 rz 7.52 deg; joints [-5.61, -27.687, 86, 93.41, 104.912, 52.654, -36.259]
  MoveL 5428 to (-57.32, 7.37, -164.49) mm, rotated rx -172.19 ry 6.28 rz 7.52 deg; joints [-5.618, -27.82, 86.275, 93.366, 104.924, 52.508, -36.259]
  MoveL 5429 to (-57.17, 5.14, -164.24) mm, rotated rx -172.19 ry 6.28 rz 7.52 deg; joints [-5.621, -27.938, 86.523, 93.328, 104.934, 52.373, -36.259]
  MoveL 5430 to (-57.02, 2.95, -164.11) mm, rotated rx -172.19 ry 6.28 rz 7.52 deg; joints [-5.626, -28.056, 86.765, 93.292, 104.943, 52.246, -36.259]
  MoveL 5431 to (-56.88, 0.82, -163.87) mm, rotated rx -172.19 ry 6.28 rz 7.52 deg; joints [-5.629, -28.167, 87, 93.256, 104.952, 52.118, -36.259]
  MoveL 5432 to (-56.73, -1.31, -163.75) mm, rotated rx -172.19 ry 6.28 rz 7.52 deg; joints [-5.633, -28.281, 87.233, 93.221, 104.961, 51.996, -36.259]
  MoveL 5433 to (-56.58, -3.44, -163.63) mm, rotated rx -172.19 ry 6.28 rz 7.52 deg; joints [-5.638, -28.396, 87.465, 93.185, 104.97, 51.874, -36.259]
  MoveL 5434 to (-56.41, -5.57, -163.39) mm, rotated rx -172.19 ry 6.28 rz 7.52 deg; joints [-5.642, -28.505, 87.698, 93.149, 104.979, 51.746, -36.259]
  MoveL 5435 to (-56.26, -7.69, -163.27) mm, rotated rx -172.19 ry 6.28 rz 7.52 deg; joints [-5.647, -28.619, 87.929, 93.113, 104.988, 51.625, -36.259]
  MoveL 5436 to (-56.1, -9.82, -163.16) mm, rotated rx -172.19 ry 6.28 rz 7.52 deg; joints [-5.652, -28.733, 88.16, 93.077, 104.997, 51.504, -36.259]
  MoveL 5437 to (-55.94, -11.95, -163.04) mm, rotated rx -172.19 ry 6.28 rz 7.52 deg; joints [-5.657, -28.846, 88.39, 93.042, 105.006, 51.383, -36.259]
  MoveL 5438 to (-55.75, -14.08, -162.81) mm, rotated rx -172.19 ry 6.28 rz 7.52 deg; joints [-5.662, -28.954, 88.62, 93.005, 105.014, 51.257, -36.259]
  MoveL 5439 to (-55.59, -16.2, -162.7) mm, rotated rx -172.19 ry 6.28 rz 7.52 deg; joints [-5.668, -29.067, 88.849, 92.969, 105.023, 51.137, -36.259]
  MoveL 5440 to (-55.4, -17.98, -162.44) mm, rotated rx -172.19 ry 6.28 rz 7.52 deg; joints [-5.672, -29.154, 89.042, 92.937, 105.031, 51.029, -36.259]
  MoveL 5441 to (-55.22, -19.62, -162.12) mm, rotated rx -172.19 ry 6.28 rz 7.52 deg; joints [-5.675, -29.231, 89.22, 92.907, 105.038, 50.924, -36.259]
  MoveL 5442 to (-55.01, -21.18, -161.7) mm, rotated rx -172.19 ry 6.28 rz 7.52 deg; joints [-5.678, -29.299, 89.389, 92.878, 105.044, 50.819, -36.259]
  MoveL 5443 to (-54.41, -19.55, -160.75) mm, rotated rx -172.19 ry 6.28 rz 7.52 deg; joints [-5.686, -29.164, 89.224, 92.879, 105.047, 50.85, -36.259]
  MoveL 5444 to (-54.41, -20.18, -160.62) mm, rotated rx -172.19 ry 6.28 rz 7.52 deg; joints [-5.685, -29.194, 89.292, 92.869, 105.048, 50.811, -36.259]
  MoveL 5445 to (-54.47, -20.76, -160.53) mm, rotated rx -172.19 ry 6.28 rz 7.52 deg; joints [-5.682, -29.224, 89.355, 92.863, 105.048, 50.778, -36.259]
  MoveL 5446 to (-54.64, -21.28, -160.5) mm, rotated rx -172.19 ry 6.28 rz 7.52 deg; joints [-5.677, -29.254, 89.41, 92.861, 105.047, 50.751, -36.259]
  MoveL 5447 to (-54.85, -21.77, -160.48) mm, rotated rx -172.19 ry 6.28 rz 7.52 deg; joints [-5.67, -29.284, 89.462, 92.861, 105.044, 50.728, -36.259]
  MoveL 5448 to (-56.67, -24.97, -160.47) mm, rotated rx -172.19 ry 6.28 rz 7.52 deg; joints [-5.611, -29.486, 89.799, 92.876, 105.022, 50.587, -36.259]
  MoveL 5449 to (-56.89, -25.37, -160.46) mm, rotated rx -172.19 ry 6.28 rz 7.52 deg; joints [-5.603, -29.511, 89.842, 92.877, 105.019, 50.568, -36.259]
  MoveL 5450 to (-57.09, -25.75, -160.43) mm, rotated rx -172.19 ry 6.28 rz 7.52 deg; joints [-5.597, -29.534, 89.882, 92.878, 105.017, 50.551, -36.259]
  MoveL 5451 to (-57.32, -26.17, -160.42) mm, rotated rx -172.19 ry 6.28 rz 7.52 deg; joints [-5.589, -29.56, 89.926, 92.88, 105.014, 50.532, -36.259]
  MoveL 5452 to (-57.58, -26.63, -160.42) mm, rotated rx -172.19 ry 6.28 rz 7.52 deg; joints [-5.581, -29.589, 89.974, 92.882, 105.011, 50.512, -36.259]
  MoveL 5453 to (-58.37, -27.99, -160.42) mm, rotated rx -172.19 ry 6.28 rz 7.52 deg; joints [-5.555, -29.675, 90.117, 92.889, 105.001, 50.453, -36.259]
  MoveL 5454 to (-58.67, -28.53, -160.4) mm, rotated rx -172.19 ry 6.28 rz 7.52 deg; joints [-5.545, -29.709, 90.174, 92.892, 104.997, 50.428, -36.259]
  MoveL 5455 to (-59, -29.17, -160.37) mm, rotated rx -172.19 ry 6.28 rz 7.52 deg; joints [-5.534, -29.747, 90.241, 92.894, 104.993, 50.398, -36.259]
  MoveL 5456 to (-59.31, -29.73, -160.34) mm, rotated rx -172.19 ry 6.28 rz 7.52 deg; joints [-5.524, -29.782, 90.301, 92.896, 104.989, 50.372, -36.259]
  MoveL 5457 to (-59.83, -30.64, -160.34) mm, rotated rx -172.19 ry 6.28 rz 7.52 deg; joints [-5.507, -29.839, 90.395, 92.901, 104.983, 50.333, -36.259]
  MoveL 5458 to (-60.62, -31.86, -160.43) mm, rotated rx -172.19 ry 6.28 rz 7.52 deg; joints [-5.482, -29.921, 90.522, 92.91, 104.973, 50.286, -36.259]
  MoveL 5459 to (-61.38, -32.77, -160.68) mm, rotated rx -172.19 ry 6.28 rz 7.52 deg; joints [-5.46, -29.991, 90.614, 92.923, 104.963, 50.262, -36.259]
  MoveL 5460 to (-62.12, -33.36, -161.1) mm, rotated rx -172.19 ry 6.28 rz 7.52 deg; joints [-5.44, -30.05, 90.672, 92.941, 104.953, 50.263, -36.259]
  MoveL 5461 to (-62.49, -33.55, -161.37) mm, rotated rx -172.19 ry 6.28 rz 7.52 deg; joints [-5.431, -30.075, 90.688, 92.951, 104.949, 50.272, -36.259]
  MoveL 5462 to (-62.85, -33.65, -161.69) mm, rotated rx -172.19 ry 6.28 rz 7.52 deg; joints [-5.423, -30.098, 90.696, 92.962, 104.944, 50.288, -36.259]
  MoveL 5463 to (-63.55, -33.62, -162.44) mm, rotated rx -172.19 ry 6.28 rz 7.52 deg; joints [-5.408, -30.135, 90.686, 92.987, 104.934, 50.336, -36.259]
  MoveL 5464 to (-64.23, -33.28, -163.37) mm, rotated rx -172.19 ry 6.28 rz 7.52 deg; joints [-5.396, -30.161, 90.641, 93.017, 104.924, 50.408, -36.259]
  MoveL 5465 to (-65.54, -31.67, -165.72) mm, rotated rx -172.19 ry 6.28 rz 7.52 deg; joints [-5.379, -30.179, 90.45, 93.087, 104.905, 50.624, -36.259]
  MoveL 5466 to (-66.4, -29.4, -168.07) mm, rotated rx -172.19 ry 6.28 rz 7.52 deg; joints [-5.376, -30.153, 90.189, 93.151, 104.891, 50.867, -36.259]
  MoveL 5467 to (-66.47, -27.06, -169.75) mm, rotated rx -172.19 ry 6.28 rz 7.52 deg; joints [-5.393, -30.087, 89.927, 93.189, 104.888, 51.07, -36.259]
  MoveL 5468 to (-66.2, -25.86, -170.34) mm, rotated rx -172.19 ry 6.28 rz 7.52 deg; joints [-5.408, -30.038, 89.795, 93.198, 104.891, 51.156, -36.259]
  MoveL 5469 to (-65.74, -24.65, -170.76) mm, rotated rx -172.19 ry 6.28 rz 7.52 deg; joints [-5.428, -29.98, 89.663, 93.201, 104.897, 51.233, -36.259]
  MoveL 5470 to (-64.21, -22.16, -171.1) mm, rotated rx -172.19 ry 6.28 rz 7.52 deg; joints [-5.481, -29.832, 89.399, 93.186, 104.918, 51.355, -36.259]
  MoveL 5471 to (-62.3, -19.66, -171.1) mm, rotated rx -172.19 ry 6.28 rz 7.52 deg; joints [-5.544, -29.666, 89.137, 93.159, 104.944, 51.456, -36.259]
  MoveL 5472 to (-61.74, -18.85, -171.14) mm, rotated rx -172.19 ry 6.28 rz 7.52 deg; joints [-5.562, -29.615, 89.051, 93.152, 104.951, 51.492, -36.259]
  MoveL 5473 to (-61.42, -18.44, -171.14) mm, rotated rx -172.19 ry 6.28 rz 7.52 deg; joints [-5.573, -29.587, 89.007, 93.147, 104.956, 51.509, -36.259]
  MoveL 5474 to (-61.1, -18.01, -171.15) mm, rotated rx -172.19 ry 6.28 rz 7.52 deg; joints [-5.583, -29.558, 88.961, 93.143, 104.96, 51.527, -36.259]
  MoveL 5475 to (-60.76, -17.55, -171.17) mm, rotated rx -172.19 ry 6.28 rz 7.52 deg; joints [-5.594, -29.529, 88.913, 93.138, 104.965, 51.547, -36.259]
  MoveL 5476 to (-60.4, -17.01, -171.23) mm, rotated rx -172.19 ry 6.28 rz 7.52 deg; joints [-5.607, -29.496, 88.855, 93.134, 104.97, 51.573, -36.259]
  MoveL 5477 to (-60.07, -16.54, -171.26) mm, rotated rx -172.19 ry 6.28 rz 7.52 deg; joints [-5.618, -29.466, 88.805, 93.13, 104.974, 51.594, -36.259]
  MoveL 5478 to (-59.76, -16.12, -171.27) mm, rotated rx -172.19 ry 6.28 rz 7.52 deg; joints [-5.628, -29.438, 88.76, 93.126, 104.979, 51.612, -36.259]
  MoveL 5479 to (-59.48, -15.72, -171.31) mm, rotated rx -172.19 ry 6.28 rz 7.52 deg; joints [-5.637, -29.413, 88.718, 93.123, 104.982, 51.631, -36.259]
  MoveL 5480 to (-59.24, -15.34, -171.35) mm, rotated rx -172.19 ry 6.28 rz 7.52 deg; joints [-5.646, -29.391, 88.677, 93.121, 104.986, 51.649, -36.259]
  MoveL 5481 to (-58.98, -14.96, -171.39) mm, rotated rx -172.19 ry 6.28 rz 7.52 deg; joints [-5.655, -29.367, 88.636, 93.118, 104.989, 51.667, -36.259]
  MoveL 5482 to (-58.68, -14.55, -171.4) mm, rotated rx -172.19 ry 6.28 rz 7.52 deg; joints [-5.664, -29.34, 88.593, 93.114, 104.993, 51.685, -36.259]
  MoveL 5483 to (-58.38, -14.14, -171.41) mm, rotated rx -172.19 ry 6.28 rz 7.52 deg; joints [-5.674, -29.313, 88.548, 93.11, 104.997, 51.703, -36.259]
  MoveL 5484 to (-58.09, -13.7, -171.42) mm, rotated rx -172.19 ry 6.28 rz 7.52 deg; joints [-5.683, -29.285, 88.502, 93.107, 105.001, 51.721, -36.259]
  MoveL 5485 to (-57.87, -13.27, -171.44) mm, rotated rx -172.19 ry 6.28 rz 7.52 deg; joints [-5.691, -29.258, 88.456, 93.106, 105.004, 51.742, -36.259]
  MoveL 5486 to (-57.71, -12.82, -171.47) mm, rotated rx -172.19 ry 6.28 rz 7.52 deg; joints [-5.696, -29.231, 88.408, 93.107, 105.006, 51.764, -36.259]
  MoveL 5487 to (-57.61, -12.38, -171.51) mm, rotated rx -172.19 ry 6.28 rz 7.52 deg; joints [-5.7, -29.207, 88.36, 93.11, 105.006, 51.789, -36.259]
  MoveL 5488 to (-57.55, -11.93, -171.56) mm, rotated rx -172.19 ry 6.28 rz 7.52 deg; joints [-5.702, -29.182, 88.311, 93.115, 105.006, 51.814, -36.259]
  MoveL 5489 to (-58.01, -13.38, -172.52) mm, rotated rx -172.19 ry 6.28 rz 7.52 deg; joints [-5.699, -29.306, 88.457, 93.112, 105.005, 51.79, -36.259]
  MoveL 5490 to (-58.07, -11.66, -172.9) mm, rotated rx -172.19 ry 6.28 rz 7.52 deg; joints [-5.7, -29.223, 88.269, 93.139, 105, 51.9, -36.259]
  MoveL 5491 to (-58.08, -9.85, -173.18) mm, rotated rx -172.19 ry 6.28 rz 7.52 deg; joints [-5.702, -29.131, 88.072, 93.166, 104.995, 52.009, -36.259]
  MoveL 5492 to (-58.04, -7.9, -173.38) mm, rotated rx -172.19 ry 6.28 rz 7.52 deg; joints [-5.704, -29.028, 87.86, 93.192, 104.991, 52.121, -36.259]
  MoveL 5493 to (-57.96, -5.77, -173.6) mm, rotated rx -172.19 ry 6.28 rz 7.52 deg; joints [-5.708, -28.913, 87.627, 93.221, 104.986, 52.243, -36.259]
  MoveL 5494 to (-57.85, -3.64, -173.72) mm, rotated rx -172.19 ry 6.28 rz 7.52 deg; joints [-5.712, -28.795, 87.395, 93.248, 104.982, 52.36, -36.259]
  MoveL 5495 to (-57.73, -1.5, -173.83) mm, rotated rx -172.19 ry 6.28 rz 7.52 deg; joints [-5.716, -28.675, 87.162, 93.275, 104.977, 52.478, -36.259]
  MoveL 5496 to (-57.63, 0.63, -174.06) mm, rotated rx -172.19 ry 6.28 rz 7.52 deg; joints [-5.72, -28.56, 86.928, 93.303, 104.973, 52.601, -36.259]
  MoveL 5497 to (-57.52, 2.76, -174.18) mm, rotated rx -172.19 ry 6.28 rz 7.52 deg; joints [-5.724, -28.441, 86.694, 93.33, 104.968, 52.719, -36.259]
  MoveL 5498 to (-57.4, 4.89, -174.3) mm, rotated rx -172.19 ry 6.28 rz 7.52 deg; joints [-5.728, -28.321, 86.46, 93.357, 104.964, 52.838, -36.259]
  MoveL 5499 to (-57.28, 7.02, -174.54) mm, rotated rx -172.19 ry 6.28 rz 7.52 deg; joints [-5.733, -28.205, 86.223, 93.385, 104.959, 52.962, -36.259]
  MoveL 5500 to (-57.15, 9.15, -174.66) mm, rotated rx -172.19 ry 6.28 rz 7.52 deg; joints [-5.738, -28.084, 85.988, 93.412, 104.955, 53.081, -36.259]
  MoveL 5501 to (-57.02, 11.28, -174.78) mm, rotated rx -172.19 ry 6.28 rz 7.52 deg; joints [-5.742, -27.963, 85.752, 93.439, 104.95, 53.201, -36.259]
  MoveL 5502 to (-56.9, 13.3, -174.97) mm, rotated rx -172.19 ry 6.28 rz 7.52 deg; joints [-5.747, -27.852, 85.527, 93.465, 104.946, 53.317, -36.259]
  MoveL 5503 to (-56.78, 15.12, -175.19) mm, rotated rx -172.19 ry 6.28 rz 7.52 deg; joints [-5.752, -27.751, 85.323, 93.489, 104.942, 53.425, -36.259]
  MoveL 5504 to (-56.65, 17.08, -175.29) mm, rotated rx -172.19 ry 6.28 rz 7.52 deg; joints [-5.756, -27.639, 85.104, 93.513, 104.938, 53.535, -36.259]
  MoveL 5505 to (-56.62, 19.25, -175.29) mm, rotated rx -172.19 ry 6.28 rz 7.52 deg; joints [-5.756, -27.512, 84.862, 93.544, 104.931, 53.654, -36.259]
  MoveL 5506 to (-56.42, 21.96, -175.38) mm, rotated rx -172.19 ry 6.28 rz 7.52 deg; joints [-5.762, -27.353, 84.558, 93.578, 104.925, 53.804, -36.259]
  MoveL 5507 to (-56.14, 24.41, -175.62) mm, rotated rx -172.19 ry 6.28 rz 7.52 deg; joints [-5.772, -27.214, 84.281, 93.606, 104.922, 53.947, -36.259]
  MoveL 5508 to (-55.99, 26.44, -175.8) mm, rotated rx -172.19 ry 6.28 rz 7.52 deg; joints [-5.777, -27.099, 84.051, 93.632, 104.918, 54.066, -36.259]
  MoveL 5509 to (-55.83, 28.3, -176.12) mm, rotated rx -172.19 ry 6.28 rz 7.52 deg; joints [-5.785, -26.998, 83.838, 93.656, 104.915, 54.182, -36.259]
  MoveL 5510 to (-55.68, 30.34, -176.3) mm, rotated rx -172.19 ry 6.28 rz 7.52 deg; joints [-5.791, -26.881, 83.605, 93.682, 104.91, 54.302, -36.259]
  MoveL 5511 to (-55.51, 32.31, -176.5) mm, rotated rx -172.19 ry 6.28 rz 7.52 deg; joints [-5.797, -26.769, 83.381, 93.707, 104.907, 54.418, -36.259]
  MoveL 5512 to (-55.31, 34.23, -176.79) mm, rotated rx -172.19 ry 6.28 rz 7.52 deg; joints [-5.805, -26.663, 83.16, 93.73, 104.904, 54.536, -36.259]
  MoveL 5513 to (-54.72, 34.92, -177.55) mm, rotated rx -172.19 ry 6.28 rz 7.52 deg; joints [-5.832, -26.64, 83.074, 93.724, 104.915, 54.603, -36.259]
  MoveL 5514 to (-54.55, 34.58, -177.93) mm, rotated rx -172.19 ry 6.28 rz 7.52 deg; joints [-5.842, -26.671, 83.109, 93.715, 104.92, 54.6, -36.259]
  MoveL 5515 to (-54.49, 34.53, -178.18) mm, rotated rx -172.19 ry 6.28 rz 7.52 deg; joints [-5.847, -26.683, 83.113, 93.713, 104.922, 54.607, -36.259]
  MoveL 5516 to (-54.55, 34.73, -178.3) mm, rotated rx -172.19 ry 6.28 rz 7.52 deg; joints [-5.847, -26.676, 83.089, 93.719, 104.921, 54.625, -36.259]
  MoveL 5517 to (-54.76, 35.21, -178.35) mm, rotated rx -172.19 ry 6.28 rz 7.52 deg; joints [-5.84, -26.651, 83.033, 93.732, 104.915, 54.657, -36.259]
  MoveL 5518 to (-55.06, 35.81, -178.39) mm, rotated rx -172.19 ry 6.28 rz 7.52 deg; joints [-5.83, -26.621, 82.964, 93.75, 104.907, 54.696, -36.259]
  MoveL 5519 to (-55.85, 37.17, -178.39) mm, rotated rx -172.19 ry 6.28 rz 7.52 deg; joints [-5.804, -26.55, 82.808, 93.795, 104.887, 54.783, -36.259]
  MoveL 5520 to (-56.12, 37.64, -178.4) mm, rotated rx -172.19 ry 6.28 rz 7.52 deg; joints [-5.795, -26.526, 82.754, 93.81, 104.88, 54.814, -36.259]
  MoveL 5521 to (-56.37, 38.11, -178.42) mm, rotated rx -172.19 ry 6.28 rz 7.52 deg; joints [-5.787, -26.502, 82.699, 93.825, 104.874, 54.845, -36.259]
  MoveL 5522 to (-56.62, 38.6, -178.47) mm, rotated rx -172.19 ry 6.28 rz 7.52 deg; joints [-5.779, -26.477, 82.642, 93.84, 104.867, 54.879, -36.259]
  MoveL 5523 to (-56.86, 39.11, -178.54) mm, rotated rx -172.19 ry 6.28 rz 7.52 deg; joints [-5.772, -26.453, 82.583, 93.855, 104.861, 54.914, -36.259]
  MoveL 5524 to (-57.1, 39.6, -178.6) mm, rotated rx -172.19 ry 6.28 rz 7.52 deg; joints [-5.765, -26.428, 82.525, 93.869, 104.855, 54.948, -36.259]
  MoveL 5525 to (-57.34, 40.04, -178.62) mm, rotated rx -172.19 ry 6.28 rz 7.52 deg; joints [-5.757, -26.406, 82.474, 93.883, 104.849, 54.977, -36.259]
  MoveL 5526 to (-57.56, 40.44, -178.64) mm, rotated rx -172.19 ry 6.28 rz 7.52 deg; joints [-5.75, -26.385, 82.428, 93.896, 104.843, 55.003, -36.259]
  MoveL 5527 to (-58.35, 41.8, -178.64) mm, rotated rx -172.19 ry 6.28 rz 7.52 deg; joints [-5.724, -26.314, 82.271, 93.94, 104.822, 55.091, -36.259]
  MoveL 5528 to (-58.6, 42.25, -178.65) mm, rotated rx -172.19 ry 6.28 rz 7.52 deg; joints [-5.716, -26.29, 82.218, 93.954, 104.816, 55.121, -36.259]
  MoveL 5529 to (-58.82, 42.67, -178.68) mm, rotated rx -172.19 ry 6.28 rz 7.52 deg; joints [-5.709, -26.269, 82.169, 93.967, 104.81, 55.149, -36.259]
  MoveL 5530 to (-59.02, 43.08, -178.73) mm, rotated rx -172.19 ry 6.28 rz 7.52 deg; joints [-5.703, -26.249, 82.122, 93.979, 104.805, 55.177, -36.259]
  MoveL 5531 to (-59.22, 43.48, -178.77) mm, rotated rx -172.19 ry 6.28 rz 7.52 deg; joints [-5.696, -26.228, 82.075, 93.992, 104.799, 55.204, -36.259]
  MoveL 5532 to (-59.46, 43.91, -178.78) mm, rotated rx -172.19 ry 6.28 rz 7.52 deg; joints [-5.689, -26.206, 82.025, 94.005, 104.793, 55.232, -36.259]
  MoveL 5533 to (-59.72, 44.36, -178.78) mm, rotated rx -172.19 ry 6.28 rz 7.52 deg; joints [-5.68, -26.182, 81.972, 94.02, 104.786, 55.262, -36.259]
  MoveL 5534 to (-60.94, 47.03, -179.12) mm, rotated rx -172.19 ry 6.28 rz 7.52 deg; joints [-5.644, -26.048, 81.658, 94.097, 104.753, 55.446, -36.259]
  MoveL 5535 to (-61.26, 48.31, -179.54) mm, rotated rx -172.19 ry 6.28 rz 7.52 deg; joints [-5.637, -25.99, 81.506, 94.127, 104.743, 55.542, -36.259]
  MoveL 5536 to (-61.38, 49.54, -180.13) mm, rotated rx -172.19 ry 6.28 rz 7.52 deg; joints [-5.639, -25.936, 81.355, 94.151, 104.737, 55.642, -36.259]
  MoveL 5537 to (-61.06, 51.91, -181.82) mm, rotated rx -172.19 ry 6.28 rz 7.52 deg; joints [-5.667, -25.846, 81.063, 94.181, 104.738, 55.852, -36.259]
  MoveL 5538 to (-59.97, 54.12, -184.19) mm, rotated rx -172.19 ry 6.28 rz 7.52 deg; joints [-5.726, -25.777, 80.782, 94.189, 104.756, 56.073, -36.259]
  MoveL 5539 to (-58.52, 55.62, -186.55) mm, rotated rx -172.19 ry 6.28 rz 7.52 deg; joints [-5.797, -25.746, 80.582, 94.176, 104.785, 56.25, -36.259]
  MoveL 5540 to (-57.82, 55.9, -187.48) mm, rotated rx -172.19 ry 6.28 rz 7.52 deg; joints [-5.83, -25.751, 80.541, 94.162, 104.8, 56.3, -36.259]
  MoveL 5541 to (-57.13, 55.86, -188.24) mm, rotated rx -172.19 ry 6.28 rz 7.52 deg; joints [-5.86, -25.771, 80.538, 94.144, 104.816, 56.324, -36.259]
  MoveL 5542 to (-56.8, 55.72, -188.55) mm, rotated rx -172.19 ry 6.28 rz 7.52 deg; joints [-5.874, -25.786, 80.551, 94.133, 104.824, 56.326, -36.259]
  MoveL 5543 to (-56.46, 55.5, -188.83) mm, rotated rx -172.19 ry 6.28 rz 7.52 deg; joints [-5.888, -25.804, 80.574, 94.12, 104.832, 56.322, -36.259]
  MoveL 5544 to (-55.81, 54.83, -189.25) mm, rotated rx -172.19 ry 6.28 rz 7.52 deg; joints [-5.914, -25.851, 80.649, 94.092, 104.849, 56.294, -36.259]
  MoveL 5545 to (-55.17, 53.84, -189.5) mm, rotated rx -172.19 ry 6.28 rz 7.52 deg; joints [-5.937, -25.912, 80.763, 94.059, 104.866, 56.241, -36.259]
  MoveL 5546 to (-54.54, 52.54, -189.59) mm, rotated rx -172.19 ry 6.28 rz 7.52 deg; joints [-5.959, -25.987, 80.916, 94.021, 104.884, 56.162, -36.259]
  MoveL 5547 to (-53.93, 51.09, -189.59) mm, rotated rx -172.19 ry 6.28 rz 7.52 deg; joints [-5.98, -26.067, 81.085, 93.981, 104.902, 56.071, -36.259]
  MoveL 5548 to (-53.73, 50.6, -189.58) mm, rotated rx -172.19 ry 6.28 rz 7.52 deg; joints [-5.986, -26.094, 81.142, 93.967, 104.908, 56.04, -36.259]
  MoveL 5549 to (-53.53, 50.06, -189.55) mm, rotated rx -172.19 ry 6.28 rz 7.52 deg; joints [-5.993, -26.124, 81.206, 93.953, 104.914, 56.005, -36.259]
  MoveL 5550 to (-53.32, 49.45, -189.48) mm, rotated rx -172.19 ry 6.28 rz 7.52 deg; joints [-5.999, -26.156, 81.278, 93.937, 104.92, 55.964, -36.259]
  MoveL 5551 to (-53.12, 48.92, -189.46) mm, rotated rx -172.19 ry 6.28 rz 7.52 deg; joints [-6.006, -26.185, 81.34, 93.923, 104.926, 55.93, -36.259]
  MoveL 5552 to (-52.92, 48.43, -189.45) mm, rotated rx -172.19 ry 6.28 rz 7.52 deg; joints [-6.012, -26.212, 81.397, 93.91, 104.932, 55.899, -36.259]
  MoveL 5553 to (-52.72, 47.95, -189.44) mm, rotated rx -172.19 ry 6.28 rz 7.52 deg; joints [-6.019, -26.238, 81.453, 93.896, 104.938, 55.869, -36.259]
  MoveL 5554 to (-52.55, 47.47, -189.4) mm, rotated rx -172.19 ry 6.28 rz 7.52 deg; joints [-6.024, -26.264, 81.51, 93.884, 104.943, 55.837, -36.259]
  MoveL 5555 to (-52.41, 46.99, -189.32) mm, rotated rx -172.19 ry 6.28 rz 7.52 deg; joints [-6.028, -26.288, 81.566, 93.872, 104.948, 55.804, -36.259]
  MoveL 5556 to (-52.27, 46.5, -189.22) mm, rotated rx -172.19 ry 6.28 rz 7.52 deg; joints [-6.032, -26.313, 81.624, 93.86, 104.952, 55.77, -36.259]
  MoveL 5557 to (-52.12, 46.02, -189.15) mm, rotated rx -172.19 ry 6.28 rz 7.52 deg; joints [-6.036, -26.338, 81.682, 93.848, 104.957, 55.737, -36.259]
  MoveL 5558 to (-51.93, 45.52, -189.12) mm, rotated rx -172.19 ry 6.28 rz 7.52 deg; joints [-6.042, -26.365, 81.739, 93.835, 104.962, 55.705, -36.259]
  MoveL 5559 to (-51.74, 45.04, -189.11) mm, rotated rx -172.19 ry 6.28 rz 7.52 deg; joints [-6.049, -26.391, 81.796, 93.822, 104.968, 55.674, -36.259]
  MoveL 5560 to (-50.78, 42.67, -189.1) mm, rotated rx -172.19 ry 6.28 rz 7.52 deg; joints [-6.081, -26.522, 82.071, 93.757, 104.996, 55.527, -36.259]
  MoveL 5561 to (-50.69, 42.29, -189.08) mm, rotated rx -172.19 ry 6.28 rz 7.52 deg; joints [-6.084, -26.543, 82.114, 93.748, 104.999, 55.503, -36.259]
  MoveL 5562 to (-50.67, 42.13, -188.96) mm, rotated rx -172.19 ry 6.28 rz 7.52 deg; joints [-6.084, -26.549, 82.135, 93.745, 104.999, 55.488, -36.259]
  MoveL 5563 to (-50.69, 42.21, -188.74) mm, rotated rx -172.19 ry 6.28 rz 7.52 deg; joints [-6.08, -26.536, 82.127, 93.746, 104.998, 55.483, -36.259]
  MoveL 5564 to (-50.75, 42.56, -188.37) mm, rotated rx -172.19 ry 6.28 rz 7.52 deg; joints [-6.074, -26.503, 82.09, 93.752, 104.994, 55.486, -36.259]
  MoveL 5565 to (-51.28, 42.01, -187.63) mm, rotated rx -172.19 ry 6.28 rz 7.52 deg; joints [-6.05, -26.518, 82.161, 93.757, 104.984, 55.428, -36.259]
  MoveL 5566 to (-51.69, 39.93, -187.61) mm, rotated rx -172.19 ry 6.28 rz 7.52 deg; joints [-6.038, -26.649, 82.401, 93.738, 104.985, 55.315, -36.259]
  MoveL 5567 to (-52.13, 37.79, -187.49) mm, rotated rx -172.19 ry 6.28 rz 7.52 deg; joints [-6.024, -26.779, 82.647, 93.718, 104.984, 55.195, -36.259]
  MoveL 5568 to (-52.63, 35.57, -187.22) mm, rotated rx -172.19 ry 6.28 rz 7.52 deg; joints [-6.006, -26.91, 82.903, 93.699, 104.983, 55.065, -36.259]
  MoveL 5569 to (-53.07, 33.5, -187.09) mm, rotated rx -172.19 ry 6.28 rz 7.52 deg; joints [-5.992, -27.035, 83.14, 93.681, 104.982, 54.949, -36.259]
  MoveL 5570 to (-53.5, 31.5, -186.83) mm, rotated rx -172.19 ry 6.28 rz 7.52 deg; joints [-5.977, -27.152, 83.37, 93.663, 104.981, 54.831, -36.259]
  MoveL 5571 to (-53.95, 29.45, -186.47) mm, rotated rx -172.19 ry 6.28 rz 7.52 deg; joints [-5.96, -27.268, 83.606, 93.645, 104.979, 54.706, -36.259]
  MoveL 5572 to (-54.38, 27.34, -186.34) mm, rotated rx -172.19 ry 6.28 rz 7.52 deg; joints [-5.947, -27.394, 83.845, 93.626, 104.979, 54.589, -36.259]
  MoveL 5573 to (-54.79, 25.27, -186.24) mm, rotated rx -172.19 ry 6.28 rz 7.52 deg; joints [-5.934, -27.519, 84.08, 93.607, 104.978, 54.476, -36.259]
  MoveL 5574 to (-55.21, 23.16, -186.09) mm, rotated rx -172.19 ry 6.28 rz 7.52 deg; joints [-5.92, -27.644, 84.318, 93.588, 104.978, 54.359, -36.259]
  MoveL 5575 to (-55.64, 21.12, -185.8) mm, rotated rx -172.19 ry 6.28 rz 7.52 deg; joints [-5.904, -27.761, 84.549, 93.571, 104.977, 54.239, -36.259]
  MoveL 5576 to (-56.02, 18.96, -185.46) mm, rotated rx -172.19 ry 6.28 rz 7.52 deg; joints [-5.89, -27.881, 84.793, 93.55, 104.976, 54.111, -36.259]
  MoveL 5577 to (-56.42, 16.88, -185.28) mm, rotated rx -172.19 ry 6.28 rz 7.52 deg; joints [-5.876, -28.002, 85.027, 93.531, 104.976, 53.994, -36.259]
  MoveL 5578 to (-56.81, 14.77, -185.17) mm, rotated rx -172.19 ry 6.28 rz 7.52 deg; joints [-5.864, -28.127, 85.262, 93.512, 104.976, 53.88, -36.259]
  MoveL 5579 to (-57.21, 12.68, -185.1) mm, rotated rx -172.19 ry 6.28 rz 7.52 deg; joints [-5.851, -28.252, 85.494, 93.494, 104.976, 53.769, -36.259]
  MoveL 5580 to (-57.59, 10.58, -184.88) mm, rotated rx -172.19 ry 6.28 rz 7.52 deg; joints [-5.838, -28.373, 85.729, 93.474, 104.975, 53.65, -36.259]
  MoveL 5581 to (-57.97, 8.49, -184.74) mm, rotated rx -172.19 ry 6.28 rz 7.52 deg; joints [-5.825, -28.495, 85.961, 93.456, 104.975, 53.536, -36.259]
  MoveL 5582 to (-58.37, 6.38, -184.66) mm, rotated rx -172.19 ry 6.28 rz 7.52 deg; joints [-5.813, -28.619, 86.193, 93.437, 104.975, 53.425, -36.259]
  MoveL 5583 to (-58.73, 4.29, -184.43) mm, rotated rx -172.19 ry 6.28 rz 7.52 deg; joints [-5.8, -28.738, 86.425, 93.418, 104.975, 53.307, -36.259]
  MoveL 5584 to (-59.08, 2.16, -184.2) mm, rotated rx -172.19 ry 6.28 rz 7.52 deg; joints [-5.787, -28.857, 86.659, 93.398, 104.975, 53.188, -36.259]
  MoveL 5585 to (-59.46, 0.02, -184.05) mm, rotated rx -172.19 ry 6.28 rz 7.52 deg; joints [-5.774, -28.98, 86.894, 93.379, 104.975, 53.072, -36.259]
  MoveL 5586 to (-59.75, -1.84, -183.93) mm, rotated rx -172.19 ry 6.28 rz 7.52 deg; joints [-5.765, -29.087, 87.097, 93.361, 104.975, 52.972, -36.259]
  MoveL 5587 to (-59.95, -3.47, -183.72) mm, rotated rx -172.19 ry 6.28 rz 7.52 deg; joints [-5.757, -29.175, 87.276, 93.343, 104.976, 52.878, -36.259]
  MoveL 5588 to (-60.05, -4.9, -183.39) mm, rotated rx -172.19 ry 6.28 rz 7.52 deg; joints [-5.751, -29.248, 87.435, 93.325, 104.978, 52.788, -36.259]
  MoveL 5589 to (-59.55, -3.51, -182.44) mm, rotated rx -172.19 ry 6.28 rz 7.52 deg; joints [-5.755, -29.127, 87.295, 93.327, 104.98, 52.809, -36.259]
  MoveL 5590 to (-59.64, -4, -182.44) mm, rotated rx -172.19 ry 6.28 rz 7.52 deg; joints [-5.752, -29.156, 87.348, 93.323, 104.979, 52.784, -36.259]
  MoveL 5591 to (-59.78, -4.48, -182.43) mm, rotated rx -172.19 ry 6.28 rz 7.52 deg; joints [-5.748, -29.185, 87.399, 93.32, 104.979, 52.76, -36.259]
  MoveL 5592 to (-60.01, -4.96, -182.41) mm, rotated rx -172.19 ry 6.28 rz 7.52 deg; joints [-5.741, -29.215, 87.451, 93.321, 104.976, 52.737, -36.259]
  MoveL 5593 to (-60.31, -5.43, -182.37) mm, rotated rx -172.19 ry 6.28 rz 7.52 deg; joints [-5.731, -29.244, 87.502, 93.323, 104.972, 52.715, -36.259]
  MoveL 5594 to (-60.68, -5.92, -182.31) mm, rotated rx -172.19 ry 6.28 rz 7.52 deg; joints [-5.718, -29.275, 87.555, 93.328, 104.966, 52.692, -36.259]
  MoveL 5595 to (-61.07, -6.35, -182.27) mm, rotated rx -172.19 ry 6.28 rz 7.52 deg; joints [-5.705, -29.304, 87.602, 93.334, 104.961, 52.673, -36.259]
  MoveL 5596 to (-61.46, -6.76, -182.26) mm, rotated rx -172.19 ry 6.28 rz 7.52 deg; joints [-5.692, -29.332, 87.646, 93.341, 104.955, 52.656, -36.259]
  MoveL 5597 to (-61.83, -7.13, -182.26) mm, rotated rx -172.19 ry 6.28 rz 7.52 deg; joints [-5.681, -29.358, 87.685, 93.347, 104.95, 52.642, -36.259]
  MoveL 5598 to (-62.19, -7.51, -182.25) mm, rotated rx -172.19 ry 6.28 rz 7.52 deg; joints [-5.669, -29.385, 87.726, 93.354, 104.944, 52.627, -36.259]
  MoveL 5599 to (-62.59, -7.95, -182.21) mm, rotated rx -172.19 ry 6.28 rz 7.52 deg; joints [-5.655, -29.414, 87.773, 93.36, 104.938, 52.608, -36.259]
  MoveL 5600 to (-63, -8.46, -182.12) mm, rotated rx -172.19 ry 6.28 rz 7.52 deg; joints [-5.641, -29.445, 87.829, 93.366, 104.932, 52.583, -36.259]
  MoveL 5601 to (-63.34, -8.85, -182.07) mm, rotated rx -172.19 ry 6.28 rz 7.52 deg; joints [-5.629, -29.47, 87.87, 93.371, 104.927, 52.565, -36.259]
  MoveL 5602 to (-63.63, -9.16, -182.05) mm, rotated rx -172.19 ry 6.28 rz 7.52 deg; joints [-5.62, -29.491, 87.904, 93.376, 104.923, 52.552, -36.259]
  MoveL 5603 to (-63.97, -9.51, -182.03) mm, rotated rx -172.19 ry 6.28 rz 7.52 deg; joints [-5.609, -29.515, 87.941, 93.381, 104.918, 52.538, -36.259]
  MoveL 5604 to (-64.33, -9.88, -182.03) mm, rotated rx -172.19 ry 6.28 rz 7.52 deg; joints [-5.597, -29.541, 87.98, 93.388, 104.912, 52.524, -36.259]
  MoveL 5605 to (-64.68, -10.24, -182.02) mm, rotated rx -172.19 ry 6.28 rz 7.52 deg; joints [-5.586, -29.566, 88.019, 93.394, 104.907, 52.509, -36.259]
  MoveL 5606 to (-65.02, -10.61, -181.99) mm, rotated rx -172.19 ry 6.28 rz 7.52 deg; joints [-5.574, -29.591, 88.059, 93.399, 104.902, 52.493, -36.259]
  MoveL 5607 to (-65.37, -10.98, -181.98) mm, rotated rx -172.19 ry 6.28 rz 7.52 deg; joints [-5.563, -29.616, 88.098, 93.406, 104.897, 52.479, -36.259]
  MoveL 5608 to (-67.23, -12.85, -181.98) mm, rotated rx -172.19 ry 6.28 rz 7.52 deg; joints [-5.502, -29.747, 88.295, 93.439, 104.87, 52.408, -36.259]
  MoveL 5609 to (-68.29, -13.83, -182.06) mm, rotated rx -172.19 ry 6.28 rz 7.52 deg; joints [-5.469, -29.821, 88.398, 93.46, 104.854, 52.377, -36.259]
  MoveL 5610 to (-69.26, -14.54, -182.31) mm, rotated rx -172.19 ry 6.28 rz 7.52 deg; joints [-5.44, -29.883, 88.469, 93.482, 104.839, 52.367, -36.259]
  MoveL 5611 to (-70.14, -14.96, -182.73) mm, rotated rx -172.19 ry 6.28 rz 7.52 deg; joints [-5.416, -29.934, 88.508, 93.505, 104.826, 52.378, -36.259]
  MoveL 5612 to (-70.91, -15.09, -183.31) mm, rotated rx -172.19 ry 6.28 rz 7.52 deg; joints [-5.397, -29.973, 88.515, 93.529, 104.814, 52.411, -36.259]
  MoveL 5613 to (-71.59, -14.95, -184.06) mm, rotated rx -172.19 ry 6.28 rz 7.52 deg; joints [-5.383, -30.001, 88.49, 93.555, 104.804, 52.465, -36.259]
  MoveL 5614 to (-72.17, -14.51, -184.97) mm, rotated rx -172.19 ry 6.28 rz 7.52 deg; joints [-5.374, -30.017, 88.433, 93.582, 104.795, 52.54, -36.259]
  MoveL 5615 to (-73.04, -12.8, -187.31) mm, rotated rx -172.19 ry 6.28 rz 7.52 deg; joints [-5.372, -30.015, 88.223, 93.639, 104.78, 52.755, -36.259]
  MoveL 5616 to (-73.33, -10.55, -189.65) mm, rotated rx -172.19 ry 6.28 rz 7.52 deg; joints [-5.388, -29.974, 87.955, 93.685, 104.774, 52.99, -36.259]
  MoveL 5617 to (-72.86, -8.33, -191.36) mm, rotated rx -172.19 ry 6.28 rz 7.52 deg; joints [-5.422, -29.902, 87.698, 93.705, 104.781, 53.182, -36.259]
  MoveL 5618 to (-72.35, -7.23, -191.97) mm, rotated rx -172.19 ry 6.28 rz 7.52 deg; joints [-5.446, -29.854, 87.574, 93.705, 104.788, 53.261, -36.259]
  MoveL 5619 to (-71.64, -6.14, -192.43) mm, rotated rx -172.19 ry 6.28 rz 7.52 deg; joints [-5.474, -29.798, 87.453, 93.699, 104.799, 53.329, -36.259]
  MoveL 5620 to (-69.67, -4, -192.86) mm, rotated rx -172.19 ry 6.28 rz 7.52 deg; joints [-5.542, -29.663, 87.22, 93.668, 104.829, 53.433, -36.259]
  MoveL 5621 to (-68.92, -3.32, -192.89) mm, rotated rx -172.19 ry 6.28 rz 7.52 deg; joints [-5.567, -29.615, 87.148, 93.654, 104.841, 53.459, -36.259]
  MoveL 5622 to (-66.85, -1.71, -192.89) mm, rotated rx -172.19 ry 6.28 rz 7.52 deg; joints [-5.634, -29.495, 86.977, 93.611, 104.873, 53.513, -36.259]
  MoveL 5623 to (-66.08, -1.06, -192.95) mm, rotated rx -172.19 ry 6.28 rz 7.52 deg; joints [-5.659, -29.449, 86.906, 93.596, 104.886, 53.539, -36.259]
  MoveL 5624 to (-65.26, -0.41, -192.95) mm, rotated rx -172.19 ry 6.28 rz 7.52 deg; joints [-5.686, -29.4, 86.837, 93.579, 104.899, 53.562, -36.259]
  MoveL 5625 to (-64.88, -0.11, -192.96) mm, rotated rx -172.19 ry 6.28 rz 7.52 deg; joints [-5.698, -29.378, 86.805, 93.572, 104.905, 53.572, -36.259]
  MoveL 5626 to (-64.55, 0.17, -192.98) mm, rotated rx -172.19 ry 6.28 rz 7.52 deg; joints [-5.709, -29.358, 86.775, 93.566, 104.91, 53.583, -36.259]
  MoveL 5627 to (-64.19, 0.46, -192.99) mm, rotated rx -172.19 ry 6.28 rz 7.52 deg; joints [-5.721, -29.337, 86.743, 93.559, 104.915, 53.594, -36.259]
  MoveL 5628 to (-62.13, 2.07, -193) mm, rotated rx -172.19 ry 6.28 rz 7.52 deg; joints [-5.787, -29.216, 86.571, 93.517, 104.948, 53.65, -36.259]
  MoveL 5629 to (-61.75, 2.39, -193.02) mm, rotated rx -172.19 ry 6.28 rz 7.52 deg; joints [-5.8, -29.193, 86.537, 93.51, 104.954, 53.662, -36.259]
  MoveL 5630 to (-61.41, 2.7, -193.06) mm, rotated rx -172.19 ry 6.28 rz 7.52 deg; joints [-5.811, -29.172, 86.502, 93.504, 104.959, 53.676, -36.259]
  MoveL 5631 to (-61.11, 3.02, -193.1) mm, rotated rx -172.19 ry 6.28 rz 7.52 deg; joints [-5.821, -29.151, 86.467, 93.499, 104.964, 53.69, -36.259]
  MoveL 5632 to (-60.84, 3.37, -193.13) mm, rotated rx -172.19 ry 6.28 rz 7.52 deg; joints [-5.83, -29.128, 86.43, 93.496, 104.968, 53.706, -36.259]
  MoveL 5633 to (-60.62, 3.75, -193.15) mm, rotated rx -172.19 ry 6.28 rz 7.52 deg; joints [-5.837, -29.104, 86.388, 93.494, 104.971, 53.724, -36.259]
  MoveL 5634 to (-60.44, 4.16, -193.15) mm, rotated rx -172.19 ry 6.28 rz 7.52 deg; joints [-5.843, -29.078, 86.344, 93.494, 104.972, 53.744, -36.259]
  MoveL 5635 to (-60.87, 3.53, -193.89) mm, rotated rx -172.19 ry 6.28 rz 7.52 deg; joints [-5.837, -29.146, 86.404, 93.501, 104.969, 53.752, -36.259]
  MoveL 5636 to (-60.67, 4.94, -194.44) mm, rotated rx -172.19 ry 6.28 rz 7.52 deg; joints [-5.849, -29.08, 86.243, 93.517, 104.97, 53.851, -36.259]
  MoveL 5637 to (-60.35, 6.47, -194.87) mm, rotated rx -172.19 ry 6.28 rz 7.52 deg; joints [-5.863, -29.002, 86.071, 93.53, 104.972, 53.948, -36.259]
  MoveL 5638 to (-59.91, 8.19, -195.17) mm, rotated rx -172.19 ry 6.28 rz 7.52 deg; joints [-5.88, -28.907, 85.879, 93.542, 104.975, 54.048, -36.259]
  MoveL 5639 to (-59.32, 10.12, -195.36) mm, rotated rx -172.19 ry 6.28 rz 7.52 deg; joints [-5.9, -28.792, 85.665, 93.552, 104.979, 54.152, -36.259]
  MoveL 5640 to (-58.7, 12.12, -195.55) mm, rotated rx -172.19 ry 6.28 rz 7.52 deg; joints [-5.921, -28.673, 85.441, 93.562, 104.984, 54.26, -36.259]
  MoveL 5641 to (-58.06, 14.15, -195.67) mm, rotated rx -172.19 ry 6.28 rz 7.52 deg; joints [-5.942, -28.549, 85.216, 93.572, 104.989, 54.366, -36.259]
  MoveL 5642 to (-57.42, 16.19, -195.9) mm, rotated rx -172.19 ry 6.28 rz 7.52 deg; joints [-5.963, -28.428, 84.988, 93.583, 104.995, 54.478, -36.259]
  MoveL 5643 to (-56.76, 18.22, -196.01) mm, rotated rx -172.19 ry 6.28 rz 7.52 deg; joints [-5.985, -28.303, 84.761, 93.593, 105, 54.584, -36.259]
  MoveL 5644 to (-56.1, 20.25, -196.13) mm, rotated rx -172.19 ry 6.28 rz 7.52 deg; joints [-6.006, -28.178, 84.533, 93.603, 105.005, 54.691, -36.259]
  MoveL 5645 to (-55.44, 22.28, -196.25) mm, rotated rx -172.19 ry 6.28 rz 7.52 deg; joints [-6.027, -28.053, 84.305, 93.613, 105.01, 54.798, -36.259]
  MoveL 5646 to (-54.78, 24.31, -196.48) mm, rotated rx -172.19 ry 6.28 rz 7.52 deg; joints [-6.049, -27.932, 84.076, 93.624, 105.016, 54.91, -36.259]
  MoveL 5647 to (-54.12, 26.34, -196.6) mm, rotated rx -172.19 ry 6.28 rz 7.52 deg; joints [-6.07, -27.806, 83.847, 93.634, 105.021, 55.018, -36.259]
  MoveL 5648 to (-53.53, 28.3, -196.71) mm, rotated rx -172.19 ry 6.28 rz 7.52 deg; joints [-6.088, -27.684, 83.624, 93.646, 105.025, 55.123, -36.259]
  MoveL 5649 to (-53.07, 30.26, -196.91) mm, rotated rx -172.19 ry 6.28 rz 7.52 deg; joints [-6.104, -27.568, 83.4, 93.662, 105.027, 55.235, -36.259]
  MoveL 5650 to (-52.26, 32.63, -197.05) mm, rotated rx -172.19 ry 6.28 rz 7.52 deg; joints [-6.13, -27.42, 83.13, 93.674, 105.033, 55.361, -36.259]
  MoveL 5651 to (-51.35, 34.91, -197.13) mm, rotated rx -172.19 ry 6.28 rz 7.52 deg; joints [-6.158, -27.273, 82.871, 93.681, 105.042, 55.479, -36.259]
  MoveL 5652 to (-50.56, 37.05, -197.17) mm, rotated rx -172.19 ry 6.28 rz 7.52 deg; joints [-6.182, -27.135, 82.626, 93.69, 105.049, 55.59, -36.259]
  MoveL 5653 to (-49.9, 39, -197.21) mm, rotated rx -172.19 ry 6.28 rz 7.52 deg; joints [-6.202, -27.01, 82.403, 93.7, 105.054, 55.692, -36.259]
  MoveL 5654 to (-49.28, 40.86, -197.33) mm, rotated rx -172.19 ry 6.28 rz 7.52 deg; joints [-6.221, -26.893, 82.188, 93.711, 105.058, 55.793, -36.259]
  MoveL 5655 to (-48.65, 42.78, -197.39) mm, rotated rx -172.19 ry 6.28 rz 7.52 deg; joints [-6.241, -26.769, 81.966, 93.721, 105.063, 55.896, -36.259]
  MoveL 5656 to (-47.97, 44.8, -197.47) mm, rotated rx -172.19 ry 6.28 rz 7.52 deg; joints [-6.261, -26.64, 81.733, 93.733, 105.068, 56.004, -36.259]
  MoveL 5657 to (-47.32, 46.68, -197.65) mm, rotated rx -172.19 ry 6.28 rz 7.52 deg; joints [-6.282, -26.523, 81.514, 93.743, 105.073, 56.11, -36.259]
  MoveL 5658 to (-46.67, 48.47, -197.96) mm, rotated rx -172.19 ry 6.28 rz 7.52 deg; joints [-6.305, -26.415, 81.303, 93.753, 105.08, 56.218, -36.259]
  MoveL 5659 to (-46, 49.03, -199) mm, rotated rx -172.19 ry 6.28 rz 7.52 deg; joints [-6.337, -26.407, 81.226, 93.745, 105.093, 56.291, -36.259]
  MoveL 5660 to (-46.03, 48.77, -199.52) mm, rotated rx -172.19 ry 6.28 rz 7.52 deg; joints [-6.342, -26.44, 81.25, 93.744, 105.096, 56.301, -36.259]
  MoveL 5661 to (-46.01, 48.75, -199.84) mm, rotated rx -172.19 ry 6.28 rz 7.52 deg; joints [-6.346, -26.452, 81.248, 93.744, 105.097, 56.315, -36.259]
  MoveL 5662 to (-45.96, 48.96, -200.01) mm, rotated rx -172.19 ry 6.28 rz 7.52 deg; joints [-6.349, -26.444, 81.222, 93.746, 105.098, 56.334, -36.259]
  MoveL 5663 to (-45.93, 49.38, -200.04) mm, rotated rx -172.19 ry 6.28 rz 7.52 deg; joints [-6.35, -26.419, 81.172, 93.752, 105.097, 56.359, -36.259]
  MoveL 5664 to (-45.94, 49.9, -200.06) mm, rotated rx -172.19 ry 6.28 rz 7.52 deg; joints [-6.349, -26.388, 81.111, 93.761, 105.094, 56.389, -36.259]
  MoveL 5665 to (-46.04, 50.49, -200.07) mm, rotated rx -172.19 ry 6.28 rz 7.52 deg; joints [-6.346, -26.353, 81.042, 93.773, 105.09, 56.425, -36.259]
  MoveL 5666 to (-46.18, 51.1, -200.08) mm, rotated rx -172.19 ry 6.28 rz 7.52 deg; joints [-6.341, -26.318, 80.971, 93.786, 105.085, 56.462, -36.259]
  MoveL 5667 to (-47.16, 54.64, -200.08) mm, rotated rx -172.19 ry 6.28 rz 7.52 deg; joints [-6.306, -26.113, 80.557, 93.87, 105.051, 56.677, -36.259]
  MoveL 5668 to (-47.27, 55.06, -200.11) mm, rotated rx -172.19 ry 6.28 rz 7.52 deg; joints [-6.303, -26.089, 80.506, 93.88, 105.047, 56.704, -36.259]
  MoveL 5669 to (-47.39, 55.53, -200.12) mm, rotated rx -172.19 ry 6.28 rz 7.52 deg; joints [-6.299, -26.062, 80.451, 93.891, 105.043, 56.733, -36.259]
  MoveL 5670 to (-47.53, 56.04, -200.13) mm, rotated rx -172.19 ry 6.28 rz 7.52 deg; joints [-6.294, -26.033, 80.391, 93.903, 105.038, 56.765, -36.259]
  MoveL 5671 to (-47.65, 56.51, -200.14) mm, rotated rx -172.19 ry 6.28 rz 7.52 deg; joints [-6.29, -26.006, 80.335, 93.914, 105.034, 56.794, -36.259]
  MoveL 5672 to (-47.75, 56.97, -200.18) mm, rotated rx -172.19 ry 6.28 rz 7.52 deg; joints [-6.287, -25.98, 80.281, 93.924, 105.03, 56.824, -36.259]
  MoveL 5673 to (-47.82, 57.39, -200.24) mm, rotated rx -172.19 ry 6.28 rz 7.52 deg; joints [-6.285, -25.957, 80.23, 93.933, 105.027, 56.852, -36.259]
  MoveL 5674 to (-47.92, 57.85, -200.28) mm, rotated rx -172.19 ry 6.28 rz 7.52 deg; joints [-6.282, -25.93, 80.175, 93.944, 105.023, 56.881, -36.259]
  MoveL 5675 to (-48.04, 58.32, -200.29) mm, rotated rx -172.19 ry 6.28 rz 7.52 deg; joints [-6.278, -25.903, 80.12, 93.955, 105.019, 56.911, -36.259]
  MoveL 5676 to (-48.17, 58.81, -200.3) mm, rotated rx -172.19 ry 6.28 rz 7.52 deg; joints [-6.273, -25.875, 80.062, 93.966, 105.014, 56.941, -36.259]
  MoveL 5677 to (-48.32, 59.31, -200.3) mm, rotated rx -172.19 ry 6.28 rz 7.52 deg; joints [-6.268, -25.846, 80.002, 93.978, 105.009, 56.972, -36.259]
  MoveL 5678 to (-48.82, 62.19, -200.64) mm, rotated rx -172.19 ry 6.28 rz 7.52 deg; joints [-6.253, -25.684, 79.657, 94.039, 104.988, 57.161, -36.259]
  MoveL 5679 to (-48.81, 63.49, -201.08) mm, rotated rx -172.19 ry 6.28 rz 7.52 deg; joints [-6.257, -25.617, 79.497, 94.06, 104.983, 57.257, -36.259]
  MoveL 5680 to (-48.62, 64.7, -201.68) mm, rotated rx -172.19 ry 6.28 rz 7.52 deg; joints [-6.269, -25.559, 79.346, 94.076, 104.984, 57.353, -36.259]
  MoveL 5681 to (-47.71, 66.85, -203.41) mm, rotated rx -172.19 ry 6.28 rz 7.52 deg; joints [-6.314, -25.469, 79.07, 94.09, 104.997, 57.548, -36.259]
  MoveL 5682 to (-46.11, 68.63, -205.84) mm, rotated rx -172.19 ry 6.28 rz 7.52 deg; joints [-6.389, -25.415, 78.828, 94.081, 105.028, 57.745, -36.259]
  MoveL 5683 to (-44.33, 69.63, -208.26) mm, rotated rx -172.19 ry 6.28 rz 7.52 deg; joints [-6.47, -25.407, 78.678, 94.055, 105.066, 57.896, -36.259]
  MoveL 5684 to (-43.59, 69.69, -209.21) mm, rotated rx -172.19 ry 6.28 rz 7.52 deg; joints [-6.504, -25.425, 78.659, 94.038, 105.084, 57.935, -36.259]
  MoveL 5685 to (-42.94, 69.45, -209.99) mm, rotated rx -172.19 ry 6.28 rz 7.52 deg; joints [-6.533, -25.456, 78.678, 94.019, 105.1, 57.949, -36.259]
  MoveL 5686 to (-42.65, 69.22, -210.31) mm, rotated rx -172.19 ry 6.28 rz 7.52 deg; joints [-6.546, -25.478, 78.702, 94.008, 105.108, 57.947, -36.259]
  MoveL 5687 to (-42.38, 68.92, -210.6) mm, rotated rx -172.19 ry 6.28 rz 7.52 deg; joints [-6.557, -25.503, 78.735, 93.996, 105.116, 57.939, -36.259]
  MoveL 5688 to (-41.91, 68.09, -211.03) mm, rotated rx -172.19 ry 6.28 rz 7.52 deg; joints [-6.578, -25.563, 78.829, 93.971, 105.13, 57.905, -36.259]
  MoveL 5689 to (-41.54, 66.96, -211.29) mm, rotated rx -172.19 ry 6.28 rz 7.52 deg; joints [-6.593, -25.638, 78.96, 93.943, 105.143, 57.847, -36.259]
  MoveL 5690 to (-41.26, 65.54, -211.37) mm, rotated rx -172.19 ry 6.28 rz 7.52 deg; joints [-6.605, -25.726, 79.129, 93.913, 105.156, 57.765, -36.259]
  MoveL 5691 to (-41.19, 65.02, -211.37) mm, rotated rx -172.19 ry 6.28 rz 7.52 deg; joints [-6.608, -25.758, 79.191, 93.902, 105.159, 57.734, -36.259]
  MoveL 5692 to (-41.14, 64.57, -211.35) mm, rotated rx -172.19 ry 6.28 rz 7.52 deg; joints [-6.609, -25.785, 79.246, 93.894, 105.162, 57.705, -36.259]
  MoveL 5693 to (-41.11, 64.14, -211.3) mm, rotated rx -172.19 ry 6.28 rz 7.52 deg; joints [-6.61, -25.81, 79.297, 93.886, 105.165, 57.678, -36.259]
  MoveL 5694 to (-41.09, 63.72, -211.24) mm, rotated rx -172.19 ry 6.28 rz 7.52 deg; joints [-6.61, -25.835, 79.348, 93.878, 105.167, 57.65, -36.259]
  MoveL 5695 to (-41.06, 63.27, -211.2) mm, rotated rx -172.19 ry 6.28 rz 7.52 deg; joints [-6.612, -25.861, 79.402, 93.87, 105.169, 57.622, -36.259]
  MoveL 5696 to (-41, 62.76, -211.19) mm, rotated rx -172.19 ry 6.28 rz 7.52 deg; joints [-6.614, -25.891, 79.463, 93.86, 105.173, 57.591, -36.259]
  MoveL 5697 to (-40.92, 62.24, -211.19) mm, rotated rx -172.19 ry 6.28 rz 7.52 deg; joints [-6.617, -25.923, 79.525, 93.849, 105.176, 57.56, -36.259]
  MoveL 5698 to (-40.85, 61.75, -211.18) mm, rotated rx -172.19 ry 6.28 rz 7.52 deg; joints [-6.62, -25.953, 79.583, 93.839, 105.18, 57.53, -36.259]
  MoveL 5699 to (-40.79, 61.28, -211.16) mm, rotated rx -172.19 ry 6.28 rz 7.52 deg; joints [-6.622, -25.981, 79.639, 93.83, 105.183, 57.501, -36.259]
  MoveL 5700 to (-40.76, 60.86, -211.1) mm, rotated rx -172.19 ry 6.28 rz 7.52 deg; joints [-6.623, -26.005, 79.69, 93.822, 105.185, 57.474, -36.259]
  MoveL 5701 to (-40.73, 60.43, -211.04) mm, rotated rx -172.19 ry 6.28 rz 7.52 deg; joints [-6.623, -26.029, 79.741, 93.814, 105.187, 57.446, -36.259]
  MoveL 5702 to (-40.7, 59.97, -210.99) mm, rotated rx -172.19 ry 6.28 rz 7.52 deg; joints [-6.624, -26.056, 79.797, 93.806, 105.19, 57.416, -36.259]
  MoveL 5703 to (-40.63, 59.36, -210.95) mm, rotated rx -172.19 ry 6.28 rz 7.52 deg; joints [-6.627, -26.092, 79.87, 93.794, 105.194, 57.378, -36.259]
  MoveL 5704 to (-40.55, 58.57, -210.93) mm, rotated rx -172.19 ry 6.28 rz 7.52 deg; joints [-6.63, -26.139, 79.963, 93.779, 105.199, 57.331, -36.259]
  MoveL 5705 to (-40.32, 57.02, -210.93) mm, rotated rx -172.19 ry 6.28 rz 7.52 deg; joints [-6.639, -26.233, 80.146, 93.748, 105.21, 57.239, -36.259]
  MoveL 5706 to (-40.21, 56.19, -210.9) mm, rotated rx -172.19 ry 6.28 rz 7.52 deg; joints [-6.643, -26.282, 80.244, 93.731, 105.215, 57.188, -36.259]
  MoveL 5707 to (-40.13, 55.57, -210.89) mm, rotated rx -172.19 ry 6.28 rz 7.52 deg; joints [-6.646, -26.319, 80.317, 93.719, 105.22, 57.151, -36.259]
  MoveL 5708 to (-40.11, 55.08, -210.88) mm, rotated rx -172.19 ry 6.28 rz 7.52 deg; joints [-6.647, -26.349, 80.375, 93.71, 105.222, 57.123, -36.259]
  MoveL 5709 to (-40.13, 54.66, -210.86) mm, rotated rx -172.19 ry 6.28 rz 7.52 deg; joints [-6.647, -26.375, 80.424, 93.704, 105.223, 57.098, -36.259]
  MoveL 5710 to (-40.18, 54.46, -210.75) mm, rotated rx -172.19 ry 6.28 rz 7.52 deg; joints [-6.644, -26.384, 80.449, 93.702, 105.223, 57.082, -36.259]
  MoveL 5711 to (-40.22, 54.52, -210.53) mm, rotated rx -172.19 ry 6.28 rz 7.52 deg; joints [-6.64, -26.374, 80.445, 93.704, 105.221, 57.075, -36.259]
  MoveL 5712 to (-40.24, 54.86, -210.18) mm, rotated rx -172.19 ry 6.28 rz 7.52 deg; joints [-6.636, -26.342, 80.41, 93.708, 105.218, 57.078, -36.259]
  MoveL 5713 to (-40.94, 54.52, -209.48) mm, rotated rx -172.19 ry 6.28 rz 7.52 deg; joints [-6.606, -26.349, 80.459, 93.72, 105.204, 57.034, -36.259]
  MoveL 5714 to (-41.84, 52.72, -209.33) mm, rotated rx -172.19 ry 6.28 rz 7.52 deg; joints [-6.578, -26.468, 80.671, 93.717, 105.193, 56.936, -36.259]
  MoveL 5715 to (-42.73, 51.02, -209.05) mm, rotated rx -172.19 ry 6.28 rz 7.52 deg; joints [-6.548, -26.576, 80.873, 93.716, 105.182, 56.837, -36.259]
  MoveL 5716 to (-43.61, 49.3, -208.77) mm, rotated rx -172.19 ry 6.28 rz 7.52 deg; joints [-6.519, -26.685, 81.078, 93.713, 105.171, 56.738, -36.259]
  MoveL 5717 to (-44.48, 47.57, -208.5) mm, rotated rx -172.19 ry 6.28 rz 7.52 deg; joints [-6.491, -26.793, 81.281, 93.711, 105.161, 56.639, -36.259]
  MoveL 5718 to (-45.39, 45.76, -208.29) mm, rotated rx -172.19 ry 6.28 rz 7.52 deg; joints [-6.461, -26.91, 81.494, 93.708, 105.15, 56.538, -36.259]
  MoveL 5719 to (-46.39, 43.89, -208.14) mm, rotated rx -172.19 ry 6.28 rz 7.52 deg; joints [-6.429, -27.033, 81.711, 93.708, 105.138, 56.439, -36.259]
  MoveL 5720 to (-47.69, 41.71, -208.04) mm, rotated rx -172.19 ry 6.28 rz 7.52 deg; joints [-6.389, -27.18, 81.963, 93.713, 105.121, 56.329, -36.259]
  MoveL 5721 to (-48.64, 39.41, -207.96) mm, rotated rx -172.19 ry 6.28 rz 7.52 deg; joints [-6.36, -27.33, 82.228, 93.705, 105.112, 56.21, -36.259]
  MoveL 5722 to (-49.45, 37.46, -207.85) mm, rotated rx -172.19 ry 6.28 rz 7.52 deg; joints [-6.335, -27.456, 82.453, 93.699, 105.104, 56.107, -36.259]
  MoveL 5723 to (-50.22, 35.73, -207.67) mm, rotated rx -172.19 ry 6.28 rz 7.52 deg; joints [-6.31, -27.566, 82.652, 93.695, 105.095, 56.012, -36.259]
  MoveL 5724 to (-51.09, 33.88, -207.54) mm, rotated rx -172.19 ry 6.28 rz 7.52 deg; joints [-6.282, -27.685, 82.864, 93.692, 105.086, 55.916, -36.259]
  MoveL 5725 to (-51.98, 32, -207.41) mm, rotated rx -172.19 ry 6.28 rz 7.52 deg; joints [-6.254, -27.806, 83.079, 93.69, 105.076, 55.818, -36.259]
  MoveL 5726 to (-52.91, 30.04, -207.34) mm, rotated rx -172.19 ry 6.28 rz 7.52 deg; joints [-6.225, -27.935, 83.302, 93.688, 105.065, 55.719, -36.259]
  MoveL 5727 to (-53.82, 28.1, -207.12) mm, rotated rx -172.19 ry 6.28 rz 7.52 deg; joints [-6.195, -28.055, 83.523, 93.686, 105.055, 55.615, -36.259]
  MoveL 5728 to (-54.73, 26.17, -207) mm, rotated rx -172.19 ry 6.28 rz 7.52 deg; joints [-6.166, -28.18, 83.741, 93.684, 105.044, 55.516, -36.259]
  MoveL 5729 to (-55.62, 24.24, -206.78) mm, rotated rx -172.19 ry 6.28 rz 7.52 deg; joints [-6.137, -28.3, 83.961, 93.681, 105.034, 55.412, -36.259]
  MoveL 5730 to (-56.53, 22.3, -206.67) mm, rotated rx -172.19 ry 6.28 rz 7.52 deg; joints [-6.108, -28.424, 84.179, 93.68, 105.024, 55.314, -36.259]
  MoveL 5731 to (-57.41, 20.36, -206.45) mm, rotated rx -172.19 ry 6.28 rz 7.52 deg; joints [-6.078, -28.545, 84.399, 93.677, 105.014, 55.211, -36.259]
  MoveL 5732 to (-58.31, 18.42, -206.34) mm, rotated rx -172.19 ry 6.28 rz 7.52 deg; joints [-6.05, -28.668, 84.615, 93.676, 105.004, 55.114, -36.259]
  MoveL 5733 to (-59.21, 16.48, -206.24) mm, rotated rx -172.19 ry 6.28 rz 7.52 deg; joints [-6.021, -28.791, 84.831, 93.675, 104.994, 55.017, -36.259]
  MoveL 5734 to (-59.96, 14.72, -206) mm, rotated rx -172.19 ry 6.28 rz 7.52 deg; joints [-5.995, -28.898, 85.029, 93.671, 104.985, 54.921, -36.259]
  MoveL 5735 to (-60.64, 13.02, -205.7) mm, rotated rx -172.19 ry 6.28 rz 7.52 deg; joints [-5.971, -28.997, 85.22, 93.666, 104.978, 54.826, -36.259]
  MoveL 5736 to (-61.26, 11.33, -205.32) mm, rotated rx -172.19 ry 6.28 rz 7.52 deg; joints [-5.948, -29.092, 85.411, 93.66, 104.971, 54.725, -36.259]
  MoveL 5737 to (-60.41, 12.47, -204.39) mm, rotated rx -172.19 ry 6.28 rz 7.52 deg; joints [-5.964, -28.982, 85.298, 93.647, 104.98, 54.729, -36.259]
  MoveL 5738 to (-60.58, 12.15, -204.33) mm, rotated rx -172.19 ry 6.28 rz 7.52 deg; joints [-5.958, -29.001, 85.334, 93.648, 104.978, 54.712, -36.259]
  MoveL 5739 to (-60.77, 11.83, -204.28) mm, rotated rx -172.19 ry 6.28 rz 7.52 deg; joints [-5.952, -29.02, 85.37, 93.649, 104.975, 54.695, -36.259]
  MoveL 5740 to (-61.05, 11.52, -204.24) mm, rotated rx -172.19 ry 6.28 rz 7.52 deg; joints [-5.943, -29.041, 85.404, 93.653, 104.971, 54.68, -36.259]
  MoveL 5741 to (-61.39, 11.23, -204.22) mm, rotated rx -172.19 ry 6.28 rz 7.52 deg; joints [-5.931, -29.062, 85.436, 93.659, 104.965, 54.669, -36.259]
  MoveL 5742 to (-61.81, 10.95, -204.21) mm, rotated rx -172.19 ry 6.28 rz 7.52 deg; joints [-5.918, -29.084, 85.467, 93.668, 104.958, 54.659, -36.259]
  MoveL 5743 to (-62.24, 10.68, -204.21) mm, rotated rx -172.19 ry 6.28 rz 7.52 deg; joints [-5.904, -29.106, 85.496, 93.677, 104.951, 54.651, -36.259]
  MoveL 5744 to (-63.15, 10.13, -204.21) mm, rotated rx -172.19 ry 6.28 rz 7.52 deg; joints [-5.875, -29.15, 85.554, 93.697, 104.936, 54.635, -36.259]
  MoveL 5745 to (-63.56, 9.87, -204.19) mm, rotated rx -172.19 ry 6.28 rz 7.52 deg; joints [-5.862, -29.17, 85.582, 93.706, 104.929, 54.626, -36.259]
  MoveL 5746 to (-63.95, 9.61, -204.14) mm, rotated rx -172.19 ry 6.28 rz 7.52 deg; joints [-5.849, -29.189, 85.612, 93.714, 104.923, 54.615, -36.259]
  MoveL 5747 to (-64.37, 9.3, -204.06) mm, rotated rx -172.19 ry 6.28 rz 7.52 deg; joints [-5.834, -29.21, 85.646, 93.722, 104.916, 54.6, -36.259]
  MoveL 5748 to (-64.85, 8.97, -204) mm, rotated rx -172.19 ry 6.28 rz 7.52 deg; joints [-5.818, -29.234, 85.683, 93.732, 104.908, 54.587, -36.259]
  MoveL 5749 to (-65.33, 8.65, -203.96) mm, rotated rx -172.19 ry 6.28 rz 7.52 deg; joints [-5.802, -29.257, 85.716, 93.742, 104.9, 54.575, -36.259]
  MoveL 5750 to (-65.79, 8.37, -203.95) mm, rotated rx -172.19 ry 6.28 rz 7.52 deg; joints [-5.788, -29.279, 85.747, 93.753, 104.892, 54.566, -36.259]
  MoveL 5751 to (-66.25, 8.1, -203.95) mm, rotated rx -172.19 ry 6.28 rz 7.52 deg; joints [-5.773, -29.302, 85.776, 93.763, 104.884, 54.558, -36.259]
  MoveL 5752 to (-67.15, 7.56, -203.95) mm, rotated rx -172.19 ry 6.28 rz 7.52 deg; joints [-5.744, -29.345, 85.834, 93.783, 104.869, 54.543, -36.259]
  MoveL 5753 to (-68.02, 7.01, -203.92) mm, rotated rx -172.19 ry 6.28 rz 7.52 deg; joints [-5.716, -29.388, 85.893, 93.802, 104.855, 54.525, -36.259]
  MoveL 5754 to (-70.27, 5.67, -203.92) mm, rotated rx -172.19 ry 6.28 rz 7.52 deg; joints [-5.643, -29.496, 86.035, 93.853, 104.817, 54.487, -36.259]
  MoveL 5755 to (-71.54, 4.99, -204.01) mm, rotated rx -172.19 ry 6.28 rz 7.52 deg; joints [-5.603, -29.556, 86.106, 93.883, 104.796, 54.474, -36.259]
  MoveL 5756 to (-72.65, 4.57, -204.27) mm, rotated rx -172.19 ry 6.28 rz 7.52 deg; joints [-5.57, -29.604, 86.146, 93.912, 104.777, 54.481, -36.259]
  MoveL 5757 to (-73.57, 4.41, -204.71) mm, rotated rx -172.19 ry 6.28 rz 7.52 deg; joints [-5.545, -29.64, 86.156, 93.939, 104.762, 54.507, -36.259]
  MoveL 5758 to (-73.97, 4.43, -205) mm, rotated rx -172.19 ry 6.28 rz 7.52 deg; joints [-5.535, -29.654, 86.15, 93.953, 104.755, 54.528, -36.259]
  MoveL 5759 to (-74.33, 4.51, -205.33) mm, rotated rx -172.19 ry 6.28 rz 7.52 deg; joints [-5.528, -29.665, 86.136, 93.966, 104.749, 54.553, -36.259]
  MoveL 5760 to (-74.9, 4.87, -206.12) mm, rotated rx -172.19 ry 6.28 rz 7.52 deg; joints [-5.518, -29.679, 86.085, 93.991, 104.739, 54.619, -36.259]
  MoveL 5761 to (-75.31, 5.5, -207.08) mm, rotated rx -172.19 ry 6.28 rz 7.52 deg; joints [-5.515, -29.681, 86.004, 94.015, 104.732, 54.705, -36.259]
  MoveL 5762 to (-75.59, 7.52, -209.54) mm, rotated rx -172.19 ry 6.28 rz 7.52 deg; joints [-5.533, -29.649, 85.75, 94.059, 104.726, 54.935, -36.259]
  MoveL 5763 to (-75.16, 9.91, -211.99) mm, rotated rx -172.19 ry 6.28 rz 7.52 deg; joints [-5.573, -29.586, 85.456, 94.086, 104.732, 55.175, -36.259]
  MoveL 5764 to (-74.03, 11.98, -213.75) mm, rotated rx -172.19 ry 6.28 rz 7.52 deg; joints [-5.629, -29.509, 85.208, 94.086, 104.751, 55.353, -36.259]
  MoveL 5765 to (-73.19, 12.9, -214.36) mm, rotated rx -172.19 ry 6.28 rz 7.52 deg; joints [-5.662, -29.464, 85.1, 94.075, 104.765, 55.419, -36.259]
  MoveL 5766 to (-72.18, 13.73, -214.8) mm, rotated rx -172.19 ry 6.28 rz 7.52 deg; joints [-5.699, -29.416, 85.004, 94.058, 104.783, 55.471, -36.259]
  MoveL 5767 to (-69.63, 15.17, -215.15) mm, rotated rx -172.19 ry 6.28 rz 7.52 deg; joints [-5.785, -29.31, 84.847, 94.001, 104.827, 55.527, -36.259]
  MoveL 5768 to (-67.22, 16.22, -215.15) mm, rotated rx -172.19 ry 6.28 rz 7.52 deg; joints [-5.862, -29.216, 84.735, 93.943, 104.87, 55.548, -36.259]
  MoveL 5769 to (-66.73, 16.42, -215.14) mm, rotated rx -172.19 ry 6.28 rz 7.52 deg; joints [-5.877, -29.197, 84.713, 93.931, 104.878, 55.552, -36.259]
  MoveL 5770 to (-66.23, 16.62, -215.11) mm, rotated rx -172.19 ry 6.28 rz 7.52 deg; joints [-5.893, -29.178, 84.693, 93.919, 104.887, 55.554, -36.259]
  MoveL 5771 to (-65.77, 16.81, -215.1) mm, rotated rx -172.19 ry 6.28 rz 7.52 deg; joints [-5.908, -29.16, 84.672, 93.908, 104.895, 55.557, -36.259]
  MoveL 5772 to (-65.37, 17, -215.12) mm, rotated rx -172.19 ry 6.28 rz 7.52 deg; joints [-5.921, -29.144, 84.652, 93.898, 104.902, 55.562, -36.259]
  MoveL 5773 to (-64.92, 17.21, -215.14) mm, rotated rx -172.19 ry 6.28 rz 7.52 deg; joints [-5.935, -29.126, 84.629, 93.888, 104.91, 55.569, -36.259]
  MoveL 5774 to (-64.41, 17.48, -215.21) mm, rotated rx -172.19 ry 6.28 rz 7.52 deg; joints [-5.952, -29.106, 84.599, 93.877, 104.919, 55.579, -36.259]
  MoveL 5775 to (-63.91, 17.76, -215.29) mm, rotated rx -172.19 ry 6.28 rz 7.52 deg; joints [-5.969, -29.085, 84.567, 93.866, 104.928, 55.591, -36.259]
  MoveL 5776 to (-63.4, 18.02, -215.34) mm, rotated rx -172.19 ry 6.28 rz 7.52 deg; joints [-5.986, -29.065, 84.539, 93.854, 104.937, 55.6, -36.259]
  MoveL 5777 to (-62.92, 18.25, -215.36) mm, rotated rx -172.19 ry 6.28 rz 7.52 deg; joints [-6.002, -29.046, 84.514, 93.843, 104.945, 55.606, -36.259]
  MoveL 5778 to (-62.45, 18.46, -215.37) mm, rotated rx -172.19 ry 6.28 rz 7.52 deg; joints [-6.017, -29.027, 84.491, 93.832, 104.954, 55.611, -36.259]
  MoveL 5779 to (-61.97, 18.67, -215.37) mm, rotated rx -172.19 ry 6.28 rz 7.52 deg; joints [-6.032, -29.008, 84.469, 93.82, 104.962, 55.616, -36.259]
  MoveL 5780 to (-61.46, 18.92, -215.4) mm, rotated rx -172.19 ry 6.28 rz 7.52 deg; joints [-6.049, -28.988, 84.441, 93.809, 104.971, 55.624, -36.259]
  MoveL 5781 to (-60.97, 19.18, -215.45) mm, rotated rx -172.19 ry 6.28 rz 7.52 deg; joints [-6.065, -28.968, 84.412, 93.798, 104.98, 55.633, -36.259]
  MoveL 5782 to (-60.49, 19.46, -215.52) mm, rotated rx -172.19 ry 6.28 rz 7.52 deg; joints [-6.081, -28.947, 84.381, 93.788, 104.988, 55.645, -36.259]
  MoveL 5783 to (-60.08, 19.76, -215.58) mm, rotated rx -172.19 ry 6.28 rz 7.52 deg; joints [-6.094, -28.926, 84.347, 93.78, 104.995, 55.658, -36.259]
  MoveL 5784 to (-59.73, 20.06, -215.61) mm, rotated rx -172.19 ry 6.28 rz 7.52 deg; joints [-6.106, -28.904, 84.313, 93.774, 105, 55.671, -36.259]
  MoveL 5785 to (-59.48, 20.37, -215.62) mm, rotated rx -172.19 ry 6.28 rz 7.52 deg; joints [-6.114, -28.882, 84.279, 93.771, 105.004, 55.685, -36.259]
  MoveL 5786 to (-59.26, 20.69, -215.62) mm, rotated rx -172.19 ry 6.28 rz 7.52 deg; joints [-6.121, -28.86, 84.243, 93.769, 105.007, 55.699, -36.259]
  MoveL 5787 to (-60.12, 19.74, -216.5) mm, rotated rx -172.19 ry 6.28 rz 7.52 deg; joints [-6.103, -28.958, 84.337, 93.784, 104.997, 55.702, -36.259]
  MoveL 5788 to (-59.36, 21.15, -216.78) mm, rotated rx -172.19 ry 6.28 rz 7.52 deg; joints [-6.13, -28.873, 84.177, 93.783, 105.007, 55.781, -36.259]
  MoveL 5789 to (-58.45, 22.71, -216.98) mm, rotated rx -172.19 ry 6.28 rz 7.52 deg; joints [-6.16, -28.774, 84.001, 93.779, 105.019, 55.862, -36.259]
  MoveL 5790 to (-57.39, 24.46, -217.11) mm, rotated rx -172.19 ry 6.28 rz 7.52 deg; joints [-6.194, -28.659, 83.803, 93.773, 105.033, 55.948, -36.259]
  MoveL 5791 to (-56.19, 26.36, -217.2) mm, rotated rx -172.19 ry 6.28 rz 7.52 deg; joints [-6.232, -28.531, 83.589, 93.766, 105.049, 56.04, -36.259]
  MoveL 5792 to (-55.07, 28.18, -217.35) mm, rotated rx -172.19 ry 6.28 rz 7.52 deg; joints [-6.268, -28.412, 83.383, 93.76, 105.064, 56.13, -36.259]
  MoveL 5793 to (-53.95, 30, -217.56) mm, rotated rx -172.19 ry 6.28 rz 7.52 deg; joints [-6.304, -28.293, 83.175, 93.754, 105.079, 56.225, -36.259]
  MoveL 5794 to (-52.88, 31.73, -217.68) mm, rotated rx -172.19 ry 6.28 rz 7.52 deg; joints [-6.338, -28.179, 82.979, 93.749, 105.093, 56.31, -36.259]
  MoveL 5795 to (-51.93, 33.31, -217.94) mm, rotated rx -172.19 ry 6.28 rz 7.52 deg; joints [-6.371, -28.079, 82.796, 93.745, 105.106, 56.397, -36.259]
  MoveL 5796 to (-50.84, 35.07, -218.16) mm, rotated rx -172.19 ry 6.28 rz 7.52 deg; joints [-6.406, -27.965, 82.594, 93.74, 105.121, 56.489, -36.259]
  MoveL 5797 to (-49.73, 36.83, -218.3) mm, rotated rx -172.19 ry 6.28 rz 7.52 deg; joints [-6.441, -27.847, 82.391, 93.735, 105.136, 56.578, -36.259]
  MoveL 5798 to (-48.58, 38.63, -218.4) mm, rotated rx -172.19 ry 6.28 rz 7.52 deg; joints [-6.477, -27.725, 82.184, 93.729, 105.151, 56.668, -36.259]
  MoveL 5799 to (-47.45, 40.43, -218.63) mm, rotated rx -172.19 ry 6.28 rz 7.52 deg; joints [-6.514, -27.607, 81.975, 93.724, 105.166, 56.763, -36.259]
  MoveL 5800 to (-46.29, 42.23, -218.89) mm, rotated rx -172.19 ry 6.28 rz 7.52 deg; joints [-6.552, -27.49, 81.765, 93.719, 105.183, 56.861, -36.259]
  MoveL 5801 to (-45.14, 44.02, -218.98) mm, rotated rx -172.19 ry 6.28 rz 7.52 deg; joints [-6.587, -27.367, 81.558, 93.713, 105.198, 56.95, -36.259]
  MoveL 5802 to (-43.97, 45.85, -219.02) mm, rotated rx -172.19 ry 6.28 rz 7.52 deg; joints [-6.623, -27.24, 81.345, 93.708, 105.213, 57.039, -36.259]
  MoveL 5803 to (-42.82, 47.63, -219.13) mm, rotated rx -172.19 ry 6.28 rz 7.52 deg; joints [-6.659, -27.118, 81.138, 93.703, 105.229, 57.129, -36.259]
  MoveL 5804 to (-41.67, 49.4, -219.33) mm, rotated rx -172.19 ry 6.28 rz 7.52 deg; joints [-6.696, -27, 80.929, 93.698, 105.244, 57.224, -36.259]
  MoveL 5805 to (-40.52, 51.14, -219.67) mm, rotated rx -172.19 ry 6.28 rz 7.52 deg; joints [-6.734, -26.887, 80.722, 93.693, 105.261, 57.323, -36.259]
  MoveL 5806 to (-39.32, 52.93, -219.92) mm, rotated rx -172.19 ry 6.28 rz 7.52 deg; joints [-6.772, -26.769, 80.51, 93.688, 105.278, 57.422, -36.259]
  MoveL 5807 to (-38.13, 54.7, -220.13) mm, rotated rx -172.19 ry 6.28 rz 7.52 deg; joints [-6.81, -26.649, 80.3, 93.682, 105.294, 57.517, -36.259]
  MoveL 5808 to (-36.91, 56.5, -220.36) mm, rotated rx -172.19 ry 6.28 rz 7.52 deg; joints [-6.849, -26.528, 80.085, 93.677, 105.311, 57.615, -36.259]
  MoveL 5809 to (-35.72, 58.29, -220.51) mm, rotated rx -172.19 ry 6.28 rz 7.52 deg; joints [-6.886, -26.404, 79.871, 93.672, 105.327, 57.71, -36.259]
  MoveL 5810 to (-34.57, 60.07, -220.53) mm, rotated rx -172.19 ry 6.28 rz 7.52 deg; joints [-6.92, -26.277, 79.66, 93.668, 105.342, 57.799, -36.259]
  MoveL 5811 to (-33.98, 60.31, -221.19) mm, rotated rx -172.19 ry 6.28 rz 7.52 deg; joints [-6.946, -26.276, 79.623, 93.658, 105.355, 57.837, -36.259]
  MoveL 5812 to (-34.09, 59.99, -221.52) mm, rotated rx -172.19 ry 6.28 rz 7.52 deg; joints [-6.947, -26.308, 79.656, 93.657, 105.355, 57.836, -36.259]
  MoveL 5813 to (-34.09, 59.95, -221.73) mm, rotated rx -172.19 ry 6.28 rz 7.52 deg; joints [-6.949, -26.317, 79.658, 93.657, 105.356, 57.843, -36.259]
  MoveL 5814 to (-34.02, 60.15, -221.83) mm, rotated rx -172.19 ry 6.28 rz 7.52 deg; joints [-6.952, -26.307, 79.632, 93.659, 105.357, 57.859, -36.259]
  MoveL 5815 to (-33.94, 60.57, -221.85) mm, rotated rx -172.19 ry 6.28 rz 7.52 deg; joints [-6.954, -26.28, 79.583, 93.664, 105.357, 57.883, -36.259]
  MoveC 5816 to (-33.9, 61.58, -221.85) mm, rotated rx -172.19 ry 6.28 rz 7.52 deg; joints [-6.954, -26.216, 79.462, 93.679, 105.353, 57.941, -36.259] to (-33.92, 62.6, -221.85) mm, rotated rx -172.19 ry 6.28 rz 7.52 deg; joints [-6.952, -26.152, 79.341, 93.696, 105.349, 58, -36.259]
  MoveL 5817 to (-33.92, 62.6, -221.86) mm, rotated rx -172.19 ry 6.28 rz 7.52 deg; joints [-6.952, -26.152, 79.341, 93.696, 105.349, 58, -36.259]
  MoveL 5818 to (-33.92, 63.14, -221.88) mm, rotated rx -172.19 ry 6.28 rz 7.52 deg; joints [-6.952, -26.119, 79.276, 93.705, 105.346, 58.033, -36.259]
  MoveL 5819 to (-33.9, 63.68, -221.93) mm, rotated rx -172.19 ry 6.28 rz 7.52 deg; joints [-6.952, -26.086, 79.211, 93.714, 105.345, 58.066, -36.259]
  MoveL 5820 to (-33.87, 64.26, -222) mm, rotated rx -172.19 ry 6.28 rz 7.52 deg; joints [-6.953, -26.051, 79.141, 93.723, 105.343, 58.103, -36.259]
  MoveL 5821 to (-33.85, 64.86, -222.04) mm, rotated rx -172.19 ry 6.28 rz 7.52 deg; joints [-6.953, -26.015, 79.07, 93.732, 105.341, 58.139, -36.259]
  MoveL 5822 to (-33.86, 66.07, -222.06) mm, rotated rx -172.19 ry 6.28 rz 7.52 deg; joints [-6.952, -25.939, 78.924, 93.752, 105.335, 58.211, -36.259]
  MoveL 5823 to (-33.85, 66.63, -222.09) mm, rotated rx -172.19 ry 6.28 rz 7.52 deg; joints [-6.952, -25.904, 78.857, 93.761, 105.333, 58.244, -36.259]
  MoveL 5824 to (-33.82, 67.1, -222.17) mm, rotated rx -172.19 ry 6.28 rz 7.52 deg; joints [-6.953, -25.876, 78.8, 93.768, 105.332, 58.275, -36.259]
  MoveL 5825 to (-33.77, 67.53, -222.26) mm, rotated rx -172.19 ry 6.28 rz 7.52 deg; joints [-6.955, -25.851, 78.746, 93.774, 105.331, 58.304, -36.259]
  MoveL 5826 to (-33.74, 67.96, -222.32) mm, rotated rx -172.19 ry 6.28 rz 7.52 deg; joints [-6.956, -25.825, 78.695, 93.781, 105.33, 58.331, -36.259]
  MoveL 5827 to (-33.73, 68.41, -222.35) mm, rotated rx -172.19 ry 6.28 rz 7.52 deg; joints [-6.956, -25.798, 78.64, 93.788, 105.328, 58.359, -36.259]
  MoveL 5828 to (-33.79, 71.03, -222.35) mm, rotated rx -172.19 ry 6.28 rz 7.52 deg; joints [-6.951, -25.632, 78.325, 93.833, 105.315, 58.513, -36.259]
  MoveL 5829 to (-33.58, 73.93, -222.7) mm, rotated rx -172.19 ry 6.28 rz 7.52 deg; joints [-6.957, -25.455, 77.97, 93.876, 105.307, 58.698, -36.259]
  MoveL 5830 to (-33.27, 75.17, -223.13) mm, rotated rx -172.19 ry 6.28 rz 7.52 deg; joints [-6.97, -25.384, 77.813, 93.89, 105.309, 58.788, -36.259]
  MoveL 5831 to (-32.82, 76.28, -223.73) mm, rotated rx -172.19 ry 6.28 rz 7.52 deg; joints [-6.989, -25.326, 77.67, 93.898, 105.315, 58.876, -36.259]
  MoveL 5832 to (-32.23, 77.25, -224.51) mm, rotated rx -172.19 ry 6.28 rz 7.52 deg; joints [-7.015, -25.28, 77.541, 93.901, 105.325, 58.964, -36.259]
  MoveL 5833 to (-31.5, 78.08, -225.46) mm, rotated rx -172.19 ry 6.28 rz 7.52 deg; joints [-7.046, -25.247, 77.426, 93.899, 105.339, 59.049, -36.259]
  MoveL 5834 to (-29.62, 79.34, -227.87) mm, rotated rx -172.19 ry 6.28 rz 7.52 deg; joints [-7.129, -25.216, 77.237, 93.878, 105.379, 59.216, -36.259]
  MoveL 5835 to (-27.77, 79.81, -230.29) mm, rotated rx -172.19 ry 6.28 rz 7.52 deg; joints [-7.211, -25.237, 77.144, 93.845, 105.422, 59.337, -36.259]
  MoveL 5836 to (-27.08, 79.65, -231.24) mm, rotated rx -172.19 ry 6.28 rz 7.52 deg; joints [-7.243, -25.267, 77.149, 93.827, 105.44, 59.365, -36.259]
  MoveL 5837 to (-26.54, 79.24, -232.01) mm, rotated rx -172.19 ry 6.28 rz 7.52 deg; joints [-7.269, -25.311, 77.188, 93.809, 105.455, 59.371, -36.259]
  MoveL 5838 to (-26.33, 78.93, -232.33) mm, rotated rx -172.19 ry 6.28 rz 7.52 deg; joints [-7.279, -25.338, 77.22, 93.799, 105.462, 59.366, -36.259]
  MoveL 5839 to (-26.16, 78.56, -232.62) mm, rotated rx -172.19 ry 6.28 rz 7.52 deg; joints [-7.288, -25.368, 77.261, 93.789, 105.468, 59.355, -36.259]
  MoveL 5840 to (-25.93, 77.63, -233.05) mm, rotated rx -172.19 ry 6.28 rz 7.52 deg; joints [-7.301, -25.438, 77.368, 93.769, 105.478, 59.318, -36.259]
  MoveL 5841 to (-25.86, 76.44, -233.31) mm, rotated rx -172.19 ry 6.28 rz 7.52 deg; joints [-7.308, -25.522, 77.51, 93.748, 105.486, 59.259, -36.259]
  MoveL 5842 to (-25.94, 74.99, -233.39) mm, rotated rx -172.19 ry 6.28 rz 7.52 deg; joints [-7.309, -25.62, 77.685, 93.726, 105.492, 59.178, -36.259]
  MoveL 5843 to (-25.99, 74.47, -233.39) mm, rotated rx -172.19 ry 6.28 rz 7.52 deg; joints [-7.308, -25.654, 77.748, 93.719, 105.493, 59.148, -36.259]
  MoveL 5844 to (-26.05, 74.02, -233.36) mm, rotated rx -172.19 ry 6.28 rz 7.52 deg; joints [-7.306, -25.683, 77.802, 93.713, 105.494, 59.121, -36.259]
  MoveL 5845 to (-26.13, 73.61, -233.3) mm, rotated rx -172.19 ry 6.28 rz 7.52 deg; joints [-7.304, -25.708, 77.853, 93.708, 105.494, 59.095, -36.259]
  MoveL 5846 to (-26.21, 73.21, -233.23) mm, rotated rx -172.19 ry 6.28 rz 7.52 deg; joints [-7.301, -25.733, 77.903, 93.703, 105.494, 59.069, -36.259]
  MoveL 5847 to (-26.29, 72.77, -233.19) mm, rotated rx -172.19 ry 6.28 rz 7.52 deg; joints [-7.299, -25.761, 77.956, 93.698, 105.494, 59.043, -36.259]
  MoveL 5848 to (-26.35, 72.27, -233.17) mm, rotated rx -172.19 ry 6.28 rz 7.52 deg; joints [-7.297, -25.793, 78.018, 93.691, 105.495, 59.013, -36.259]
  MoveL 5849 to (-26.92, 66.57, -233.16) mm, rotated rx -172.19 ry 6.28 rz 7.52 deg; joints [-7.288, -26.165, 78.704, 93.611, 105.509, 58.687, -36.259]
  MoveL 5850 to (-27.01, 65.81, -233.15) mm, rotated rx -172.19 ry 6.28 rz 7.52 deg; joints [-7.286, -26.214, 78.795, 93.601, 105.511, 58.643, -36.259]
  MoveL 5851 to (-27.12, 65.16, -233.14) mm, rotated rx -172.19 ry 6.28 rz 7.52 deg; joints [-7.283, -26.257, 78.873, 93.593, 105.512, 58.606, -36.259]
  MoveL 5852 to (-27.29, 64.61, -233.12) mm, rotated rx -172.19 ry 6.28 rz 7.52 deg; joints [-7.278, -26.294, 78.939, 93.589, 105.51, 58.576, -36.259]
  MoveL 5853 to (-27.53, 64.13, -233.08) mm, rotated rx -172.19 ry 6.28 rz 7.52 deg; joints [-7.271, -26.327, 78.998, 93.587, 105.508, 58.549, -36.259]
  MoveL 5854 to (-27.72, 63.86, -232.92) mm, rotated rx -172.19 ry 6.28 rz 7.52 deg; joints [-7.264, -26.341, 79.032, 93.588, 105.505, 58.528, -36.259]
  MoveL 5855 to (-27.74, 63.87, -232.61) mm, rotated rx -172.19 ry 6.28 rz 7.52 deg; joints [-7.26, -26.331, 79.035, 93.587, 105.503, 58.514, -36.259]
  MoveL 5856 to (-27.57, 64.2, -232.13) mm, rotated rx -172.19 ry 6.28 rz 7.52 deg; joints [-7.26, -26.293, 79.004, 93.586, 105.503, 58.507, -36.259]
  MoveL 5857 to (-28.19, 64.29, -231.16) mm, rotated rx -172.19 ry 6.28 rz 7.52 deg; joints [-7.23, -26.264, 79.007, 93.6, 105.487, 58.473, -36.259]
  MoveL 5858 to (-29.42, 62.87, -230.86) mm, rotated rx -172.19 ry 6.28 rz 7.52 deg; joints [-7.19, -26.361, 79.181, 93.61, 105.468, 58.392, -36.259]
  MoveL 5859 to (-30.69, 61.38, -230.65) mm, rotated rx -172.19 ry 6.28 rz 7.52 deg; joints [-7.15, -26.466, 79.362, 93.621, 105.449, 58.312, -36.259]
  MoveL 5860 to (-32.05, 59.75, -230.52) mm, rotated rx -172.19 ry 6.28 rz 7.52 deg; joints [-7.108, -26.584, 79.557, 93.633, 105.428, 58.23, -36.259]
  MoveL 5861 to (-34.77, 56.46, -230.52) mm, rotated rx -172.19 ry 6.28 rz 7.52 deg; joints [-7.026, -26.828, 79.947, 93.657, 105.389, 58.075, -36.259]
  MoveL 5862 to (-36.03, 54.93, -230.44) mm, rotated rx -172.19 ry 6.28 rz 7.52 deg; joints [-6.988, -26.938, 80.129, 93.668, 105.37, 58, -36.259]
  MoveL 5863 to (-37.39, 53.28, -230.44) mm, rotated rx -172.19 ry 6.28 rz 7.52 deg; joints [-6.947, -27.06, 80.322, 93.68, 105.35, 57.924, -36.259]
  MoveL 5864 to (-38.84, 51.68, -230.44) mm, rotated rx -172.19 ry 6.28 rz 7.52 deg; joints [-6.903, -27.179, 80.51, 93.696, 105.328, 57.852, -36.259]
  MoveL 5865 to (-40.57, 49.82, -230.26) mm, rotated rx -172.19 ry 6.28 rz 7.52 deg; joints [-6.848, -27.313, 80.729, 93.716, 105.301, 57.761, -36.259]
  MoveL 5866 to (-41.89, 48.02, -230.02) mm, rotated rx -172.19 ry 6.28 rz 7.52 deg; joints [-6.806, -27.435, 80.942, 93.725, 105.282, 57.666, -36.259]
  MoveL 5867 to (-43.19, 46.29, -229.9) mm, rotated rx -172.19 ry 6.28 rz 7.52 deg; joints [-6.766, -27.556, 81.145, 93.735, 105.264, 57.579, -36.259]
  MoveL 5868 to (-44.55, 44.64, -229.8) mm, rotated rx -172.19 ry 6.28 rz 7.52 deg; joints [-6.723, -27.673, 81.337, 93.748, 105.243, 57.5, -36.259]
  MoveL 5869 to (-45.9, 42.99, -229.58) mm, rotated rx -172.19 ry 6.28 rz 7.52 deg; joints [-6.68, -27.787, 81.53, 93.761, 105.223, 57.415, -36.259]
  MoveL 5870 to (-47.25, 41.34, -229.47) mm, rotated rx -172.19 ry 6.28 rz 7.52 deg; joints [-6.638, -27.903, 81.722, 93.774, 105.203, 57.336, -36.259]
  MoveL 5871 to (-48.6, 39.69, -229.36) mm, rotated rx -172.19 ry 6.28 rz 7.52 deg; joints [-6.595, -28.019, 81.912, 93.788, 105.183, 57.258, -36.259]
  MoveL 5872 to (-49.94, 38.03, -229.15) mm, rotated rx -172.19 ry 6.28 rz 7.52 deg; joints [-6.552, -28.132, 82.105, 93.801, 105.163, 57.174, -36.259]
  MoveL 5873 to (-51.29, 36.37, -229.05) mm, rotated rx -172.19 ry 6.28 rz 7.52 deg; joints [-6.51, -28.248, 82.295, 93.814, 105.143, 57.096, -36.259]
  MoveL 5874 to (-52.63, 34.72, -228.94) mm, rotated rx -172.19 ry 6.28 rz 7.52 deg; joints [-6.467, -28.364, 82.484, 93.829, 105.123, 57.018, -36.259]
  MoveL 5875 to (-53.96, 33.05, -228.73) mm, rotated rx -172.19 ry 6.28 rz 7.52 deg; joints [-6.424, -28.477, 82.676, 93.842, 105.103, 56.934, -36.259]
  MoveL 5876 to (-55.31, 31.39, -228.63) mm, rotated rx -172.19 ry 6.28 rz 7.52 deg; joints [-6.382, -28.593, 82.865, 93.856, 105.083, 56.857, -36.259]
  MoveL 5877 to (-56.41, 29.9, -228.37) mm, rotated rx -172.19 ry 6.28 rz 7.52 deg; joints [-6.345, -28.69, 83.036, 93.866, 105.067, 56.779, -36.259]
  MoveL 5878 to (-57.36, 28.53, -228.01) mm, rotated rx -172.19 ry 6.28 rz 7.52 deg; joints [-6.312, -28.774, 83.196, 93.872, 105.053, 56.7, -36.259]
  MoveL 5879 to (-58.17, 27.24, -227.51) mm, rotated rx -172.19 ry 6.28 rz 7.52 deg; joints [-6.282, -28.846, 83.348, 93.875, 105.041, 56.616, -36.259]
  MoveL 5880 to (-57.27, 27.93, -226.66) mm, rotated rx -172.19 ry 6.28 rz 7.52 deg; joints [-6.301, -28.765, 83.283, 93.855, 105.053, 56.6, -36.259]
  MoveL 5881 to (-57.48, 27.68, -226.63) mm, rotated rx -172.19 ry 6.28 rz 7.52 deg; joints [-6.294, -28.782, 83.311, 93.858, 105.049, 56.588, -36.259]
  MoveL 5882 to (-57.71, 27.45, -226.59) mm, rotated rx -172.19 ry 6.28 rz 7.52 deg; joints [-6.286, -28.797, 83.337, 93.861, 105.046, 56.577, -36.259]
  MoveL 5883 to (-58.03, 27.26, -226.54) mm, rotated rx -172.19 ry 6.28 rz 7.52 deg; joints [-6.276, -28.811, 83.359, 93.867, 105.04, 56.568, -36.259]
  MoveL 5884 to (-58.4, 27.08, -226.5) mm, rotated rx -172.19 ry 6.28 rz 7.52 deg; joints [-6.263, -28.826, 83.379, 93.876, 105.033, 56.562, -36.259]
  MoveL 5885 to (-58.86, 26.91, -226.47) mm, rotated rx -172.19 ry 6.28 rz 7.52 deg; joints [-6.248, -28.841, 83.398, 93.887, 105.025, 56.558, -36.259]
  MoveL 5886 to (-63.37, 25.56, -226.47) mm, rotated rx -172.19 ry 6.28 rz 7.52 deg; joints [-6.105, -28.982, 83.543, 94.001, 104.942, 56.548, -36.259]
